(* PLC project Adressering.ecp, WAGO e!COCKPIT e!COCKPIT *)
(* stored: creationDateTime 2021-01-18T14:20:23.2110188, modificationDateTime 2021-01-18T11:51:27.6823754 *)

TYPE dtRomtype_11111111111111 : STRUCT
  RB601_V : BOOL;  (* Bevegelse *)
  RB601_HVAC : BOOL;  (* HVAC signal *)
  RT601_CT : REAL;  (* Rom temperatur *)
  RT601_SP_D : REAL;  (* Temperatur SP *)
  RT601_SP_S : REAL;  (* Temperatur SP standby *)
  RT601_SP_N : REAL;  (* Temperatur SP nattsenk *)
  RT601_SP_F : REAL;  (* Temperatur SP frostsikring *)
  RT601_CS : REAL;  (* Aktivt temperatur SP *)
  OPM : INT;  (* Rom modus *)
  OPM_CV : INT;  (* Rom modus verdi *)
  RY601_CV : REAL;  (* Co2 Nivaa *)
  RY601_SP : REAL;  (* Co2 SP *)
  RY601_OP : REAL;  (* Co2 paadrag *)
  LH601_OP : REAL;  (* Varmepaadrag *)
  LH601_MAN : BOOL;  (* Force LH *)
  LH601_CMD : BOOL;  (* LH601_CMD *)
  LC601_OP : REAL;  (* LC601_OP *)
  LC601_SP : REAL;  (* LC SP *)
  LC601_MAN : BOOL;  (* Force LC *)
  LC601_CMD : BOOL;  (* LC601_CMD *)
  RT601_SP : REAL;  (* Temperatur SP feedback *)
  RT601_SP_FB : REAL;  (* Temperatur SP *)
  RT601_SP_IN : REAL;  (* Temperatur SP lokalt panel *)
  LU601_V : BOOL;  (* Befukter status *)
  LU601_AL : BOOL;  (* Befukter alarm/feil *)
  LU601_CMD : BOOL;  (* Befukter tillat start *)
  OPM_001 : BYTE;  (* OPM output *)
END_STRUCT;
END_TYPE

TYPE dtRomtype_33333333333333 : STRUCT
  RB601_V : BOOL;  (* Bevegelse *)
  RB602_V : BOOL;  (* Bevegelse *)
  RB603_V : BOOL;  (* Bevegelse *)
  RB601_HVAC : BOOL;  (* HVAC signal *)
  RB602_HVAC : BOOL;  (* HVAC signal *)
  RB603_HVAC : BOOL;  (* HVAC signal *)
  RT601_CT : REAL;  (* Rom temperatur *)
  RT602_CT : REAL;  (* Rom temperatur *)
  RT602_SP : REAL;  (* Temperatur SP *)
  RT603_CT : REAL;  (* Rom temperatur *)
  RT603_SP : REAL;  (* Temperatur SP *)
  RT601_SP_D : REAL;  (* Temperatur SP *)
  RT601_SP_S : REAL;  (* Temperatur SP standby *)
  RT601_SP_N : REAL;  (* Temperatur SP nattsenk *)
  RT601_SP_F : REAL;  (* Temperatur SP frostsikring *)
  RT601_CS : REAL;  (* Aktivt temperatur SP *)
  OPM : INT;  (* Rom modus *)
  OPM_CV : INT;  (* Rom modus verdi *)
  RY601_CV : REAL;  (* Co2 Nivaa *)
  RY602_CV : REAL;  (* Co2 Nivaa *)
  RY603_CV : REAL;  (* Co2 Nivaa *)
  RY601_SP : REAL;  (* Co2 SP *)
  RY601_OP : REAL;  (* Co2 paadrag *)
  LH601_OP : REAL;  (* Varmepaadrag *)
  LH602_OP : REAL;  (* Varmepaadrag *)
  LH603_OP : REAL;  (* Varmepaadrag *)
  LH601_MAN : BOOL;  (* Force LH *)
  LH601_CMD : BOOL;  (* LH601_CMD *)
  LH602_CMD : BOOL;  (* LH602_CMD *)
  LH603_CMD : BOOL;  (* LH603_CMD *)
  LC601_OP : REAL;  (* LC601_OP *)
  LC602_OP : REAL;  (* LC602_OP *)
  LC603_OP : REAL;  (* LC603_OP *)
  LC601_SP : REAL;  (* LC SP *)
  LC601_MAN : BOOL;  (* Force LC *)
  LC601_CMD : BOOL;  (* LC601_CMD *)
  LC602_CMD : BOOL;  (* LC602_CMD *)
  LC603_CMD : BOOL;  (* LC603_CMD *)
  RT601_SP : REAL;  (* Temperatur SP feedback *)
  RT601_SP_FB : REAL;  (* Temperatur SP *)
  RT601_SP_IN : REAL;  (* Temperatur SP lokalt panel *)
  RT602_SP_FB : REAL;  (* Temperatur SP *)
  RT602_SP_IN : REAL;  (* Temperatur SP lokalt panel *)
  RT603_SP_FB : REAL;  (* Temperatur SP *)
  RT603_SP_IN : REAL;  (* Temperatur SP lokalt panel *)
  LU601_V : BOOL;  (* Befukter status *)
  LU602_V : BOOL;  (* Befukter status *)
  LU603_V : BOOL;  (* Befukter status *)
  LU601_AL : BOOL;  (* Befukter alarm/feil *)
  LU602_AL : BOOL;  (* Befukter alarm/feil *)
  LU603_AL : BOOL;  (* Befukter alarm/feil *)
  LU601_CMD : BOOL;  (* Befukter tillat start *)
  LU602_CMD : BOOL;  (* Befukter tillat start *)
  LU603_CMD : BOOL;  (* Befukter tillat start *)
  OPM_001 : BYTE;  (* OPM output *)
  OPM_002 : BYTE;  (* OPM output *)
  OPM_003 : BYTE;  (* OPM output *)
END_STRUCT;
END_TYPE

TYPE dtRomtype_99999999999999 : STRUCT
  RB601_V : BOOL;  (* Bevegelse *)
  RB602_V : BOOL;  (* Bevegelse *)
  RB603_V : BOOL;  (* Bevegelse *)
  RB604_V : BOOL;  (* Bevegelse *)
  RB605_V : BOOL;  (* Bevegelse *)
  RB606_V : BOOL;  (* Bevegelse *)
  RB607_V : BOOL;  (* Bevegelse *)
  RB608_V : BOOL;  (* Bevegelse *)
  RB609_V : BOOL;  (* Bevegelse *)
  RB601_HVAC : BOOL;  (* HVAC signal *)
  RB602_HVAC : BOOL;  (* HVAC signal *)
  RB603_HVAC : BOOL;  (* HVAC signal *)
  RB604_HVAC : BOOL;  (* HVAC signal *)
  RB605_HVAC : BOOL;  (* HVAC signal *)
  RB606_HVAC : BOOL;  (* HVAC signal *)
  RB607_HVAC : BOOL;  (* HVAC signal *)
  RB608_HVAC : BOOL;  (* HVAC signal *)
  RB609_HVAC : BOOL;  (* HVAC signal *)
  RT601_CT : REAL;  (* Rom temperatur *)
  RT602_CT : REAL;  (* Rom temperatur *)
  RT602_SP : REAL;  (* Temperatur SP *)
  RT603_CT : REAL;  (* Rom temperatur *)
  RT603_SP : REAL;  (* Temperatur SP *)
  RT604_CT : REAL;  (* Rom temperatur *)
  RT604_SP : REAL;  (* Temperatur SP *)
  RT605_CT : REAL;  (* Rom temperatur *)
  RT605_SP : REAL;  (* Temperatur SP *)
  RT606_CT : REAL;  (* Rom temperatur *)
  RT606_SP : REAL;  (* Temperatur SP *)
  RT607_CT : REAL;  (* Rom temperatur *)
  RT607_SP : REAL;  (* Temperatur SP *)
  RT608_CT : REAL;  (* Rom temperatur *)
  RT608_SP : REAL;  (* Temperatur SP *)
  RT609_CT : REAL;  (* Rom temperatur *)
  RT609_SP : REAL;  (* Temperatur SP *)
  RT601_SP_D : REAL;  (* Temperatur SP *)
  RT601_SP_S : REAL;  (* Temperatur SP standby *)
  RT601_SP_N : REAL;  (* Temperatur SP nattsenk *)
  RT601_SP_F : REAL;  (* Temperatur SP frostsikring *)
  RT601_CS : REAL;  (* Aktivt temperatur SP *)
  OPM : INT;  (* Rom modus *)
  OPM_CV : INT;  (* Rom modus verdi *)
  RY601_CV : REAL;  (* Co2 Nivaa *)
  RY602_CV : REAL;  (* Co2 Nivaa *)
  RY603_CV : REAL;  (* Co2 Nivaa *)
  RY604_CV : REAL;  (* Co2 Nivaa *)
  RY605_CV : REAL;  (* Co2 Nivaa *)
  RY606_CV : REAL;  (* Co2 Nivaa *)
  RY607_CV : REAL;  (* Co2 Nivaa *)
  RY608_CV : REAL;  (* Co2 Nivaa *)
  RY609_CV : REAL;  (* Co2 Nivaa *)
  RY601_SP : REAL;  (* Co2 SP *)
  RY601_OP : REAL;  (* Co2 paadrag *)
  LH601_OP : REAL;  (* Varmepaadrag *)
  LH602_OP : REAL;  (* Varmepaadrag *)
  LH603_OP : REAL;  (* Varmepaadrag *)
  LH604_OP : REAL;  (* Varmepaadrag *)
  LH605_OP : REAL;  (* Varmepaadrag *)
  LH606_OP : REAL;  (* Varmepaadrag *)
  LH607_OP : REAL;  (* Varmepaadrag *)
  LH608_OP : REAL;  (* Varmepaadrag *)
  LH609_OP : REAL;  (* Varmepaadrag *)
  LH601_MAN : BOOL;  (* Force LH *)
  LH601_CMD : BOOL;  (* LH601_CMD *)
  LH602_CMD : BOOL;  (* LH602_CMD *)
  LH603_CMD : BOOL;  (* LH603_CMD *)
  LH604_CMD : BOOL;  (* LH604_CMD *)
  LH605_CMD : BOOL;  (* LH605_CMD *)
  LH606_CMD : BOOL;  (* LH606_CMD *)
  LH607_CMD : BOOL;  (* LH607_CMD *)
  LH608_CMD : BOOL;  (* LH608_CMD *)
  LH609_CMD : BOOL;  (* LH609_CMD *)
  LC601_OP : REAL;  (* LC601_OP *)
  LC602_OP : REAL;  (* LC602_OP *)
  LC603_OP : REAL;  (* LC603_OP *)
  LC604_OP : REAL;  (* LC604_OP *)
  LC605_OP : REAL;  (* LC605_OP *)
  LC606_OP : REAL;  (* LC606_OP *)
  LC607_OP : REAL;  (* LC607_OP *)
  LC608_OP : REAL;  (* LC608_OP *)
  LC609_OP : REAL;  (* LC609_OP *)
  LC601_SP : REAL;  (* LC SP *)
  LC601_MAN : BOOL;  (* Force LC *)
  LC601_CMD : BOOL;  (* LC601_CMD *)
  LC602_CMD : BOOL;  (* LC602_CMD *)
  LC603_CMD : BOOL;  (* LC603_CMD *)
  LC604_CMD : BOOL;  (* LC604_CMD *)
  LC605_CMD : BOOL;  (* LC605_CMD *)
  LC606_CMD : BOOL;  (* LC606_CMD *)
  LC607_CMD : BOOL;  (* LC607_CMD *)
  LC608_CMD : BOOL;  (* LC608_CMD *)
  LC609_CMD : BOOL;  (* LC609_CMD *)
  RT601_SP : REAL;  (* Temperatur SP feedback *)
  RT601_SP_FB : REAL;  (* Temperatur SP *)
  RT601_SP_IN : REAL;  (* Temperatur SP lokalt panel *)
  RT602_SP_FB : REAL;  (* Temperatur SP *)
  RT602_SP_IN : REAL;  (* Temperatur SP lokalt panel *)
  RT603_SP_FB : REAL;  (* Temperatur SP *)
  RT603_SP_IN : REAL;  (* Temperatur SP lokalt panel *)
  RT604_SP_FB : REAL;  (* Temperatur SP *)
  RT604_SP_IN : REAL;  (* Temperatur SP lokalt panel *)
  RT605_SP_FB : REAL;  (* Temperatur SP *)
  RT605_SP_IN : REAL;  (* Temperatur SP lokalt panel *)
  RT606_SP_FB : REAL;  (* Temperatur SP *)
  RT606_SP_IN : REAL;  (* Temperatur SP lokalt panel *)
  RT607_SP_FB : REAL;  (* Temperatur SP *)
  RT607_SP_IN : REAL;  (* Temperatur SP lokalt panel *)
  RT608_SP_FB : REAL;  (* Temperatur SP *)
  RT608_SP_IN : REAL;  (* Temperatur SP lokalt panel *)
  RT609_SP_FB : REAL;  (* Temperatur SP *)
  RT609_SP_IN : REAL;  (* Temperatur SP lokalt panel *)
  LU601_V : BOOL;  (* Befukter status *)
  LU602_V : BOOL;  (* Befukter status *)
  LU603_V : BOOL;  (* Befukter status *)
  LU604_V : BOOL;  (* Befukter status *)
  LU605_V : BOOL;  (* Befukter status *)
  LU606_V : BOOL;  (* Befukter status *)
  LU607_V : BOOL;  (* Befukter status *)
  LU608_V : BOOL;  (* Befukter status *)
  LU609_V : BOOL;  (* Befukter status *)
  LU601_AL : BOOL;  (* Befukter alarm/feil *)
  LU602_AL : BOOL;  (* Befukter alarm/feil *)
  LU603_AL : BOOL;  (* Befukter alarm/feil *)
  LU604_AL : BOOL;  (* Befukter alarm/feil *)
  LU605_AL : BOOL;  (* Befukter alarm/feil *)
  LU606_AL : BOOL;  (* Befukter alarm/feil *)
  LU607_AL : BOOL;  (* Befukter alarm/feil *)
  LU608_AL : BOOL;  (* Befukter alarm/feil *)
  LU609_AL : BOOL;  (* Befukter alarm/feil *)
  LU601_CMD : BOOL;  (* Befukter tillat start *)
  LU602_CMD : BOOL;  (* Befukter tillat start *)
  LU603_CMD : BOOL;  (* Befukter tillat start *)
  LU604_CMD : BOOL;  (* Befukter tillat start *)
  LU605_CMD : BOOL;  (* Befukter tillat start *)
  LU606_CMD : BOOL;  (* Befukter tillat start *)
  LU607_CMD : BOOL;  (* Befukter tillat start *)
  LU608_CMD : BOOL;  (* Befukter tillat start *)
  LU609_CMD : BOOL;  (* Befukter tillat start *)
  OPM_001 : BYTE;  (* OPM output *)
  OPM_002 : BYTE;  (* OPM output *)
  OPM_003 : BYTE;  (* OPM output *)
  OPM_004 : BYTE;  (* OPM output *)
  OPM_005 : BYTE;  (* OPM output *)
  OPM_006 : BYTE;  (* OPM output *)
  OPM_007 : BYTE;  (* OPM output *)
  OPM_008 : BYTE;  (* OPM output *)
  OPM_009 : BYTE;  (* OPM output *)
END_STRUCT;
END_TYPE

{attribute 'qualified_only'}
VAR_GLOBAL  (* STLV59_563 *)
  STLV59_A_563_RB001_HVAC : BOOL;  (* HVAC signal for PLS *)
  STLV59_A_563_KNX_Card_1_Status : BOOL;  (* KNX kort 1 status *)
  STLV59_A_563_001 : dtRomtype_11111111111111;  (* Placeholder_1 *)
  STLV59_A_563_002 : dtRomtype_33333333333333;  (* Placeholder_2 *)
  STLV59_A_563_003 : dtRomtype_99999999999999;  (* Placeholder_3 *)
END_VAR

FUNCTION_BLOCK fbRomtype_11111111111111
  VAR_INPUT
    RB601_HVAC : BOOL;
    RT601_CT : REAL;
    RT601_SP_D : REAL;
    RT601_SP_S : REAL;
    RT601_SP_N : REAL;
    RT601_SP_F : REAL;
    OPM : INT;
    RY601_CV : REAL;
    RY601_SP : REAL;
    LH601_MAN : BOOL;
    LC601_SP : REAL;
    LC601_MAN : BOOL;
    RT601_SP_IN : REAL;
    LU601_V : BOOL;
  END_VAR
  VAR_OUTPUT
    OPM_CV : INT;
    RT601_CS : REAL;
    RY601_OP : REAL;
    LH601_OP : REAL;
    LH601_CMD : BOOL;
    LC601_OP : REAL;
    LC601_CMD : BOOL;
    LU601_CMD : BOOL;
    OPM_001 : BYTE;
  END_VAR

(* CFC diagram, written out as Structured Text *)
END_FUNCTION_BLOCK

FUNCTION_BLOCK fbRomtype_33333333333333
  VAR_INPUT
    RB601_HVAC : BOOL;
    RB602_HVAC : BOOL;
    RB603_HVAC : BOOL;
    RT601_CT : REAL;
    RT602_CT : REAL;
    RT602_SP : REAL;
    RT603_CT : REAL;
    RT603_SP : REAL;
    RT601_SP_D : REAL;
    RT601_SP_S : REAL;
    RT601_SP_N : REAL;
    RT601_SP_F : REAL;
    OPM : INT;
    RY601_CV : REAL;
    RY602_CV : REAL;
    RY603_CV : REAL;
    RY601_SP : REAL;
    LH601_MAN : BOOL;
    LC601_SP : REAL;
    LC601_MAN : BOOL;
    RT601_SP_IN : REAL;
    RT602_SP_IN : REAL;
    RT603_SP_IN : REAL;
    LU601_V : BOOL;
    LU602_V : BOOL;
    LU603_V : BOOL;
  END_VAR
  VAR_OUTPUT
    OPM_CV : INT;
    RT601_CS : REAL;
    RT602_CS : REAL;
    RT603_CS : REAL;
    RY601_OP : REAL;
    LH601_OP : REAL;
    LH602_OP : REAL;
    LH603_OP : REAL;
    LH601_CMD : BOOL;
    LH602_CMD : BOOL;
    LH603_CMD : BOOL;
    LC601_OP : REAL;
    LC602_OP : REAL;
    LC603_OP : REAL;
    LC601_CMD : BOOL;
    LC602_CMD : BOOL;
    LC603_CMD : BOOL;
    LU601_CMD : BOOL;
    LU602_CMD : BOOL;
    LU603_CMD : BOOL;
    OPM_001 : BYTE;
    OPM_002 : BYTE;
    OPM_003 : BYTE;
  END_VAR

(* CFC diagram, written out as Structured Text *)
END_FUNCTION_BLOCK

FUNCTION_BLOCK fbRomtype_99999999999999
  VAR_INPUT
    RB601_HVAC : BOOL;
    RB602_HVAC : BOOL;
    RB603_HVAC : BOOL;
    RB604_HVAC : BOOL;
    RB605_HVAC : BOOL;
    RB606_HVAC : BOOL;
    RB607_HVAC : BOOL;
    RB608_HVAC : BOOL;
    RB609_HVAC : BOOL;
    RT601_CT : REAL;
    RT602_CT : REAL;
    RT602_SP : REAL;
    RT603_CT : REAL;
    RT603_SP : REAL;
    RT604_CT : REAL;
    RT604_SP : REAL;
    RT605_CT : REAL;
    RT605_SP : REAL;
    RT606_CT : REAL;
    RT606_SP : REAL;
    RT607_CT : REAL;
    RT607_SP : REAL;
    RT608_CT : REAL;
    RT608_SP : REAL;
    RT609_CT : REAL;
    RT609_SP : REAL;
    RT601_SP_D : REAL;
    RT601_SP_S : REAL;
    RT601_SP_N : REAL;
    RT601_SP_F : REAL;
    OPM : INT;
    RY601_CV : REAL;
    RY602_CV : REAL;
    RY603_CV : REAL;
    RY604_CV : REAL;
    RY605_CV : REAL;
    RY606_CV : REAL;
    RY607_CV : REAL;
    RY608_CV : REAL;
    RY609_CV : REAL;
    RY601_SP : REAL;
    LH601_MAN : BOOL;
    LC601_SP : REAL;
    LC601_MAN : BOOL;
    RT601_SP_IN : REAL;
    RT602_SP_IN : REAL;
    RT603_SP_IN : REAL;
    RT604_SP_IN : REAL;
    RT605_SP_IN : REAL;
    RT606_SP_IN : REAL;
    RT607_SP_IN : REAL;
    RT608_SP_IN : REAL;
    RT609_SP_IN : REAL;
    LU601_V : BOOL;
    LU602_V : BOOL;
    LU603_V : BOOL;
    LU604_V : BOOL;
    LU605_V : BOOL;
    LU606_V : BOOL;
    LU607_V : BOOL;
    LU608_V : BOOL;
    LU609_V : BOOL;
  END_VAR
  VAR_OUTPUT
    OPM_CV : INT;
    RT601_CS : REAL;
    RT602_CS : REAL;
    RT603_CS : REAL;
    RT604_CS : REAL;
    RT605_CS : REAL;
    RT606_CS : REAL;
    RT607_CS : REAL;
    RT608_CS : REAL;
    RT609_CS : REAL;
    RY601_OP : REAL;
    LH601_OP : REAL;
    LH602_OP : REAL;
    LH603_OP : REAL;
    LH604_OP : REAL;
    LH605_OP : REAL;
    LH606_OP : REAL;
    LH607_OP : REAL;
    LH608_OP : REAL;
    LH609_OP : REAL;
    LH601_CMD : BOOL;
    LH602_CMD : BOOL;
    LH603_CMD : BOOL;
    LH604_CMD : BOOL;
    LH605_CMD : BOOL;
    LH606_CMD : BOOL;
    LH607_CMD : BOOL;
    LH608_CMD : BOOL;
    LH609_CMD : BOOL;
    LC601_OP : REAL;
    LC602_OP : REAL;
    LC603_OP : REAL;
    LC604_OP : REAL;
    LC605_OP : REAL;
    LC606_OP : REAL;
    LC607_OP : REAL;
    LC608_OP : REAL;
    LC609_OP : REAL;
    LC601_CMD : BOOL;
    LC602_CMD : BOOL;
    LC603_CMD : BOOL;
    LC604_CMD : BOOL;
    LC605_CMD : BOOL;
    LC606_CMD : BOOL;
    LC607_CMD : BOOL;
    LC608_CMD : BOOL;
    LC609_CMD : BOOL;
    LU601_CMD : BOOL;
    LU602_CMD : BOOL;
    LU603_CMD : BOOL;
    LU604_CMD : BOOL;
    LU605_CMD : BOOL;
    LU606_CMD : BOOL;
    LU607_CMD : BOOL;
    LU608_CMD : BOOL;
    LU609_CMD : BOOL;
    OPM_001 : BYTE;
    OPM_002 : BYTE;
    OPM_003 : BYTE;
    OPM_004 : BYTE;
    OPM_005 : BYTE;
    OPM_006 : BYTE;
    OPM_007 : BYTE;
    OPM_008 : BYTE;
    OPM_009 : BYTE;
  END_VAR

(* CFC diagram, written out as Structured Text *)
END_FUNCTION_BLOCK

PROGRAM PRG_KNX_563_1
  VAR
    i : INT := 0;  (* Felles *)
    Interval : TON := (PT := TIME#2m0s0ms);
    typDPT : typDPT;
    KNX_master_1 : WagoAppKNX.FbKNX_Master;  (* Master *)
    M1_001_001_RB601_V : fbDPT_Switch_pro;  (* 001 *)
    M1_002_001_RB601_HVAC : fbDPT_Switch_pro;
    M1_003_001_RT601_CT : fbDPT_Value_Temp_pro;
    M1_004_001_RY601_CV : fbDPT_Value_AirQuality_pro;
    M1_005_001_LH601_OP : fbDPT_Scaling_pro;
    M1_006_001_LH601_CMD : fbDPT_Switch_pro;
    M1_007_001_LC601_OP : fbDPT_Scaling_pro;
    M1_008_001_LC601_CMD : fbDPT_Switch_pro;
    M1_009_001_RT601_SP : fbDPT_Value_Temp_pro;
    M1_010_001_RT601_SP_FB : fbDPT_Value_Temp_pro;
    M1_011_001_LU601_V : fbDPT_Switch_pro;
    M1_012_001_LU601_AL : fbDPT_Switch_pro;
    M1_013_001_LU601_CMD : fbDPT_Switch_pro;
    M1_014_001_OPM_001 : fbDPT_1_BYTE;
    M1_015_002_RB601_V : fbDPT_Switch_pro;  (* 002 *)
    M1_016_002_RB602_V : fbDPT_Switch_pro;
    M1_017_002_RB603_V : fbDPT_Switch_pro;
    M1_018_002_RB601_HVAC : fbDPT_Switch_pro;
    M1_019_002_RB602_HVAC : fbDPT_Switch_pro;
    M1_020_002_RB603_HVAC : fbDPT_Switch_pro;
    M1_021_002_RT601_CT : fbDPT_Value_Temp_pro;
    M1_022_002_RT602_CT : fbDPT_Value_Temp_pro;
    M1_023_002_RT603_CT : fbDPT_Value_Temp_pro;
    M1_024_002_RY601_CV : fbDPT_Value_AirQuality_pro;
    M1_025_002_RY602_CV : fbDPT_Value_AirQuality_pro;
    M1_026_002_RY603_CV : fbDPT_Value_AirQuality_pro;
    M1_027_002_LH601_OP : fbDPT_Scaling_pro;
    M1_028_002_LH602_OP : fbDPT_Scaling_pro;
    M1_029_002_LH603_OP : fbDPT_Scaling_pro;
    M1_030_002_LH601_CMD : fbDPT_Switch_pro;
    M1_031_002_LH602_CMD : fbDPT_Switch_pro;
    M1_032_002_LH603_CMD : fbDPT_Switch_pro;
    M1_033_002_LC601_OP : fbDPT_Scaling_pro;
    M1_034_002_LC602_OP : fbDPT_Scaling_pro;
    M1_035_002_LC603_OP : fbDPT_Scaling_pro;
    M1_036_002_LC601_CMD : fbDPT_Switch_pro;
    M1_037_002_LC602_CMD : fbDPT_Switch_pro;
    M1_038_002_LC603_CMD : fbDPT_Switch_pro;
    M1_039_002_RT601_SP : fbDPT_Value_Temp_pro;
    M1_040_002_RT602_SP : fbDPT_Value_Temp_pro;
    M1_041_002_RT603_SP : fbDPT_Value_Temp_pro;
    M1_042_002_RT601_SP_FB : fbDPT_Value_Temp_pro;
    M1_043_002_RT602_SP_FB : fbDPT_Value_Temp_pro;
    M1_044_002_RT603_SP_FB : fbDPT_Value_Temp_pro;
    M1_045_002_LU601_V : fbDPT_Switch_pro;
    M1_046_002_LU602_V : fbDPT_Switch_pro;
    M1_047_002_LU603_V : fbDPT_Switch_pro;
    M1_048_002_LU601_AL : fbDPT_Switch_pro;
    M1_049_002_LU602_AL : fbDPT_Switch_pro;
    M1_050_002_LU603_AL : fbDPT_Switch_pro;
    M1_051_002_LU601_CMD : fbDPT_Switch_pro;
    M1_052_002_LU602_CMD : fbDPT_Switch_pro;
    M1_053_002_LU603_CMD : fbDPT_Switch_pro;
    M1_054_002_OPM_001 : fbDPT_1_BYTE;
    M1_055_002_OPM_002 : fbDPT_1_BYTE;
    M1_056_002_OPM_003 : fbDPT_1_BYTE;
    M1_057_003_RB601_V : fbDPT_Switch_pro;  (* 003 *)
    M1_058_003_RB602_V : fbDPT_Switch_pro;
    M1_059_003_RB603_V : fbDPT_Switch_pro;
    M1_060_003_RB604_V : fbDPT_Switch_pro;
    M1_061_003_RB605_V : fbDPT_Switch_pro;
    M1_062_003_RB606_V : fbDPT_Switch_pro;
    M1_063_003_RB607_V : fbDPT_Switch_pro;
    M1_064_003_RB608_V : fbDPT_Switch_pro;
    M1_065_003_RB609_V : fbDPT_Switch_pro;
    M1_066_003_RB601_HVAC : fbDPT_Switch_pro;
    M1_067_003_RB602_HVAC : fbDPT_Switch_pro;
    M1_068_003_RB603_HVAC : fbDPT_Switch_pro;
    M1_069_003_RB604_HVAC : fbDPT_Switch_pro;
    M1_070_003_RB605_HVAC : fbDPT_Switch_pro;
    M1_071_003_RB606_HVAC : fbDPT_Switch_pro;
    M1_072_003_RB607_HVAC : fbDPT_Switch_pro;
    M1_073_003_RB608_HVAC : fbDPT_Switch_pro;
    M1_074_003_RB609_HVAC : fbDPT_Switch_pro;
    M1_075_003_RT601_CT : fbDPT_Value_Temp_pro;
    M1_076_003_RT602_CT : fbDPT_Value_Temp_pro;
    M1_077_003_RT603_CT : fbDPT_Value_Temp_pro;
    M1_078_003_RT604_CT : fbDPT_Value_Temp_pro;
    M1_079_003_RT605_CT : fbDPT_Value_Temp_pro;
    M1_080_003_RT606_CT : fbDPT_Value_Temp_pro;
    M1_081_003_RT607_CT : fbDPT_Value_Temp_pro;
    M1_082_003_RT608_CT : fbDPT_Value_Temp_pro;
    M1_083_003_RT609_CT : fbDPT_Value_Temp_pro;
    M1_084_003_RY601_CV : fbDPT_Value_AirQuality_pro;
    M1_085_003_RY602_CV : fbDPT_Value_AirQuality_pro;
    M1_086_003_RY603_CV : fbDPT_Value_AirQuality_pro;
    M1_087_003_RY604_CV : fbDPT_Value_AirQuality_pro;
    M1_088_003_RY605_CV : fbDPT_Value_AirQuality_pro;
    M1_089_003_RY606_CV : fbDPT_Value_AirQuality_pro;
    M1_090_003_RY607_CV : fbDPT_Value_AirQuality_pro;
    M1_091_003_RY608_CV : fbDPT_Value_AirQuality_pro;
    M1_092_003_RY609_CV : fbDPT_Value_AirQuality_pro;
    M1_093_003_LH601_OP : fbDPT_Scaling_pro;
    M1_094_003_LH602_OP : fbDPT_Scaling_pro;
    M1_095_003_LH603_OP : fbDPT_Scaling_pro;
    M1_096_003_LH604_OP : fbDPT_Scaling_pro;
    M1_097_003_LH605_OP : fbDPT_Scaling_pro;
    M1_098_003_LH606_OP : fbDPT_Scaling_pro;
    M1_099_003_LH607_OP : fbDPT_Scaling_pro;
    M1_0100_003_LH608_OP : fbDPT_Scaling_pro;
    M1_0101_003_LH609_OP : fbDPT_Scaling_pro;
    M1_102_003_LH601_CMD : fbDPT_Switch_pro;
    M1_103_003_LH602_CMD : fbDPT_Switch_pro;
    M1_104_003_LH603_CMD : fbDPT_Switch_pro;
    M1_105_003_LH604_CMD : fbDPT_Switch_pro;
    M1_106_003_LH605_CMD : fbDPT_Switch_pro;
    M1_107_003_LH606_CMD : fbDPT_Switch_pro;
    M1_108_003_LH607_CMD : fbDPT_Switch_pro;
    M1_109_003_LH608_CMD : fbDPT_Switch_pro;
    M1_110_003_LH609_CMD : fbDPT_Switch_pro;
    M1_111_003_LC601_OP : fbDPT_Scaling_pro;
    M1_112_003_LC602_OP : fbDPT_Scaling_pro;
    M1_113_003_LC603_OP : fbDPT_Scaling_pro;
    M1_114_003_LC604_OP : fbDPT_Scaling_pro;
    M1_115_003_LC605_OP : fbDPT_Scaling_pro;
    M1_116_003_LC606_OP : fbDPT_Scaling_pro;
    M1_117_003_LC607_OP : fbDPT_Scaling_pro;
    M1_118_003_LC608_OP : fbDPT_Scaling_pro;
    M1_119_003_LC609_OP : fbDPT_Scaling_pro;
    M1_120_003_LC601_CMD : fbDPT_Switch_pro;
    M1_121_003_LC602_CMD : fbDPT_Switch_pro;
    M1_122_003_LC603_CMD : fbDPT_Switch_pro;
    M1_123_003_LC604_CMD : fbDPT_Switch_pro;
    M1_124_003_LC605_CMD : fbDPT_Switch_pro;
    M1_125_003_LC606_CMD : fbDPT_Switch_pro;
    M1_126_003_LC607_CMD : fbDPT_Switch_pro;
    M1_127_003_LC608_CMD : fbDPT_Switch_pro;
    M1_128_003_LC609_CMD : fbDPT_Switch_pro;
    M1_129_003_RT601_SP : fbDPT_Value_Temp_pro;
    M1_130_003_RT602_SP : fbDPT_Value_Temp_pro;
    M1_131_003_RT603_SP : fbDPT_Value_Temp_pro;
    M1_132_003_RT604_SP : fbDPT_Value_Temp_pro;
    M1_133_003_RT605_SP : fbDPT_Value_Temp_pro;
    M1_134_003_RT606_SP : fbDPT_Value_Temp_pro;
    M1_135_003_RT607_SP : fbDPT_Value_Temp_pro;
    M1_136_003_RT608_SP : fbDPT_Value_Temp_pro;
    M1_137_003_RT609_SP : fbDPT_Value_Temp_pro;
    M1_138_003_RT601_SP_FB : fbDPT_Value_Temp_pro;
    M1_139_003_RT602_SP_FB : fbDPT_Value_Temp_pro;
    M1_140_003_RT603_SP_FB : fbDPT_Value_Temp_pro;
    M1_141_003_RT604_SP_FB : fbDPT_Value_Temp_pro;
    M1_142_003_RT605_SP_FB : fbDPT_Value_Temp_pro;
    M1_143_003_RT606_SP_FB : fbDPT_Value_Temp_pro;
    M1_144_003_RT607_SP_FB : fbDPT_Value_Temp_pro;
    M1_145_003_RT608_SP_FB : fbDPT_Value_Temp_pro;
    M1_146_003_RT609_SP_FB : fbDPT_Value_Temp_pro;
    M1_147_003_LU601_V : fbDPT_Switch_pro;
    M1_148_003_LU602_V : fbDPT_Switch_pro;
    M1_149_003_LU603_V : fbDPT_Switch_pro;
    M1_150_003_LU604_V : fbDPT_Switch_pro;
    M1_151_003_LU605_V : fbDPT_Switch_pro;
    M1_152_003_LU606_V : fbDPT_Switch_pro;
    M1_153_003_LU607_V : fbDPT_Switch_pro;
    M1_154_003_LU608_V : fbDPT_Switch_pro;
    M1_155_003_LU609_V : fbDPT_Switch_pro;
    M1_156_003_LU601_AL : fbDPT_Switch_pro;
    M1_157_003_LU602_AL : fbDPT_Switch_pro;
    M1_158_003_LU603_AL : fbDPT_Switch_pro;
    M1_159_003_LU604_AL : fbDPT_Switch_pro;
    M1_160_003_LU605_AL : fbDPT_Switch_pro;
    M1_161_003_LU606_AL : fbDPT_Switch_pro;
    M1_162_003_LU607_AL : fbDPT_Switch_pro;
    M1_163_003_LU608_AL : fbDPT_Switch_pro;
    M1_164_003_LU609_AL : fbDPT_Switch_pro;
    M1_165_003_LU601_CMD : fbDPT_Switch_pro;
    M1_166_003_LU602_CMD : fbDPT_Switch_pro;
    M1_167_003_LU603_CMD : fbDPT_Switch_pro;
    M1_168_003_LU604_CMD : fbDPT_Switch_pro;
    M1_169_003_LU605_CMD : fbDPT_Switch_pro;
    M1_170_003_LU606_CMD : fbDPT_Switch_pro;
    M1_171_003_LU607_CMD : fbDPT_Switch_pro;
    M1_172_003_LU608_CMD : fbDPT_Switch_pro;
    M1_173_003_LU609_CMD : fbDPT_Switch_pro;
    M1_174_003_OPM_001 : fbDPT_1_BYTE;
    M1_175_003_OPM_002 : fbDPT_1_BYTE;
    M1_176_003_OPM_003 : fbDPT_1_BYTE;
    M1_177_003_OPM_004 : fbDPT_1_BYTE;
    M1_178_003_OPM_005 : fbDPT_1_BYTE;
    M1_179_003_OPM_006 : fbDPT_1_BYTE;
    M1_180_003_OPM_007 : fbDPT_1_BYTE;
    M1_181_003_OPM_008 : fbDPT_1_BYTE;
    M1_182_003_OPM_009 : fbDPT_1_BYTE;
  END_VAR
  VAR  (* added by the conversion: wires and edge detectors of the diagram *)
    _ADD9_OUT : INT;
    _GT15_OUT : BOOL;
    _MOVE19_ENO : BOOL;
    _MOVE19_OUT : INT;
    _MOVE46_ENO : BOOL;
    _MOVE46_OUT : ANY;
    _MOVE59_ENO : BOOL;
    _MOVE59_OUT : ANY;
    _MOVE72_ENO : BOOL;
    _MOVE72_OUT : ANY;
    _MOVE85_ENO : BOOL;
    _MOVE85_OUT : ANY;
    _MOVE174_ENO : BOOL;
    _MOVE174_OUT : ANY;
    _MOVE187_ENO : BOOL;
    _MOVE187_OUT : ANY;
    _MOVE200_ENO : BOOL;
    _MOVE200_OUT : ANY;
    _MOVE246_ENO : BOOL;
    _MOVE246_OUT : ANY;
    _MOVE259_ENO : BOOL;
    _MOVE259_OUT : ANY;
    _MOVE272_ENO : BOOL;
    _MOVE272_OUT : ANY;
    _MOVE285_ENO : BOOL;
    _MOVE285_OUT : ANY;
    _MOVE298_ENO : BOOL;
    _MOVE298_OUT : ANY;
    _MOVE311_ENO : BOOL;
    _MOVE311_OUT : ANY;
    _MOVE324_ENO : BOOL;
    _MOVE324_OUT : ANY;
    _MOVE337_ENO : BOOL;
    _MOVE337_OUT : ANY;
    _MOVE350_ENO : BOOL;
    _MOVE350_OUT : ANY;
    _MOVE363_ENO : BOOL;
    _MOVE363_OUT : ANY;
    _MOVE376_ENO : BOOL;
    _MOVE376_OUT : ANY;
    _MOVE389_ENO : BOOL;
    _MOVE389_OUT : ANY;
    _MOVE630_ENO : BOOL;
    _MOVE630_OUT : ANY;
    _MOVE643_ENO : BOOL;
    _MOVE643_OUT : ANY;
    _MOVE656_ENO : BOOL;
    _MOVE656_OUT : ANY;
    _MOVE669_ENO : BOOL;
    _MOVE669_OUT : ANY;
    _MOVE682_ENO : BOOL;
    _MOVE682_OUT : ANY;
    _MOVE695_ENO : BOOL;
    _MOVE695_OUT : ANY;
    _MOVE708_ENO : BOOL;
    _MOVE708_OUT : ANY;
    _MOVE721_ENO : BOOL;
    _MOVE721_OUT : ANY;
    _MOVE734_ENO : BOOL;
    _MOVE734_OUT : ANY;
    _MOVE844_ENO : BOOL;
    _MOVE844_OUT : ANY;
    _MOVE857_ENO : BOOL;
    _MOVE857_OUT : ANY;
    _MOVE870_ENO : BOOL;
    _MOVE870_OUT : ANY;
    _MOVE883_ENO : BOOL;
    _MOVE883_OUT : ANY;
    _MOVE896_ENO : BOOL;
    _MOVE896_OUT : ANY;
    _MOVE909_ENO : BOOL;
    _MOVE909_OUT : ANY;
    _MOVE922_ENO : BOOL;
    _MOVE922_OUT : ANY;
    _MOVE935_ENO : BOOL;
    _MOVE935_OUT : ANY;
    _MOVE948_ENO : BOOL;
    _MOVE948_OUT : ANY;
    _MOVE961_ENO : BOOL;
    _MOVE961_OUT : ANY;
    _MOVE974_ENO : BOOL;
    _MOVE974_OUT : ANY;
    _MOVE987_ENO : BOOL;
    _MOVE987_OUT : ANY;
    _MOVE1000_ENO : BOOL;
    _MOVE1000_OUT : ANY;
    _MOVE1013_ENO : BOOL;
    _MOVE1013_OUT : ANY;
    _MOVE1026_ENO : BOOL;
    _MOVE1026_OUT : ANY;
    _MOVE1039_ENO : BOOL;
    _MOVE1039_OUT : ANY;
    _MOVE1052_ENO : BOOL;
    _MOVE1052_OUT : ANY;
    _MOVE1065_ENO : BOOL;
    _MOVE1065_OUT : ANY;
    _MOVE1078_ENO : BOOL;
    _MOVE1078_OUT : ANY;
    _MOVE1091_ENO : BOOL;
    _MOVE1091_OUT : ANY;
    _MOVE1104_ENO : BOOL;
    _MOVE1104_OUT : ANY;
    _MOVE1117_ENO : BOOL;
    _MOVE1117_OUT : ANY;
    _MOVE1130_ENO : BOOL;
    _MOVE1130_OUT : ANY;
    _MOVE1143_ENO : BOOL;
    _MOVE1143_OUT : ANY;
    _MOVE1156_ENO : BOOL;
    _MOVE1156_OUT : ANY;
    _MOVE1169_ENO : BOOL;
    _MOVE1169_OUT : ANY;
    _MOVE1182_ENO : BOOL;
    _MOVE1182_OUT : ANY;
    _MOVE1195_ENO : BOOL;
    _MOVE1195_OUT : ANY;
    _MOVE1208_ENO : BOOL;
    _MOVE1208_OUT : ANY;
    _MOVE1221_ENO : BOOL;
    _MOVE1221_OUT : ANY;
    _MOVE1234_ENO : BOOL;
    _MOVE1234_OUT : ANY;
    _MOVE1247_ENO : BOOL;
    _MOVE1247_OUT : ANY;
    _MOVE1260_ENO : BOOL;
    _MOVE1260_OUT : ANY;
    _MOVE1273_ENO : BOOL;
    _MOVE1273_OUT : ANY;
    _MOVE1286_ENO : BOOL;
    _MOVE1286_OUT : ANY;
    _MOVE1299_ENO : BOOL;
    _MOVE1299_OUT : ANY;
    _MOVE1996_ENO : BOOL;
    _MOVE1996_OUT : ANY;
    _MOVE2009_ENO : BOOL;
    _MOVE2009_OUT : ANY;
    _MOVE2022_ENO : BOOL;
    _MOVE2022_OUT : ANY;
    _MOVE2035_ENO : BOOL;
    _MOVE2035_OUT : ANY;
    _MOVE2048_ENO : BOOL;
    _MOVE2048_OUT : ANY;
    _MOVE2061_ENO : BOOL;
    _MOVE2061_OUT : ANY;
    _MOVE2074_ENO : BOOL;
    _MOVE2074_OUT : ANY;
    _MOVE2087_ENO : BOOL;
    _MOVE2087_OUT : ANY;
    _MOVE2100_ENO : BOOL;
    _MOVE2100_OUT : ANY;
    _MOVE2113_ENO : BOOL;
    _MOVE2113_OUT : ANY;
    _MOVE2126_ENO : BOOL;
    _MOVE2126_OUT : ANY;
    _MOVE2139_ENO : BOOL;
    _MOVE2139_OUT : ANY;
    _MOVE2152_ENO : BOOL;
    _MOVE2152_OUT : ANY;
    _MOVE2165_ENO : BOOL;
    _MOVE2165_OUT : ANY;
    _MOVE2178_ENO : BOOL;
    _MOVE2178_OUT : ANY;
    _MOVE2191_ENO : BOOL;
    _MOVE2191_OUT : ANY;
    _MOVE2204_ENO : BOOL;
    _MOVE2204_OUT : ANY;
    _MOVE2217_ENO : BOOL;
    _MOVE2217_OUT : ANY;
    _MOVE2230_ENO : BOOL;
    _MOVE2230_OUT : ANY;
    _MOVE2243_ENO : BOOL;
    _MOVE2243_OUT : ANY;
    _MOVE2256_ENO : BOOL;
    _MOVE2256_OUT : ANY;
    _MOVE2269_ENO : BOOL;
    _MOVE2269_OUT : ANY;
    _MOVE2282_ENO : BOOL;
    _MOVE2282_OUT : ANY;
    _MOVE2295_ENO : BOOL;
    _MOVE2295_OUT : ANY;
    _MOVE2308_ENO : BOOL;
    _MOVE2308_OUT : ANY;
    _MOVE2321_ENO : BOOL;
    _MOVE2321_OUT : ANY;
    _MOVE2334_ENO : BOOL;
    _MOVE2334_OUT : ANY;
  END_VAR

(* CFC diagram, written out as Structured Text *)
(* KNX Sending interval *)
(* KNX Master *)
Interval(IN := Interval.Q);
_ADD9_OUT := BOOL_TO_INT(Interval.Q) + i;
i := _ADD9_OUT;
_GT15_OUT := i > 77;
_MOVE19_OUT := MOVE(EN := _GT15_OUT, IN := 0, ENO => _MOVE19_ENO);
IF _MOVE19_ENO THEN i := _MOVE19_OUT; END_IF;
KNX_master_1(I_Port := IoConfig_Globals.KNX_EIB_TP1_Interface, bPortKNX := 1);
STLV59_563.STLV59_A_563_KNX_Card_1_Status := KNX_master_1.sStatus = 'OK';
(* Rom 001 *)
(* RB601_V *)
(* RB601_HVAC *)
M1_001_001_RB601_V(bPortKNX := 1, dwIndex_DPT := 1, typDPT := typDPT);
_MOVE46_OUT := MOVE(EN := M1_001_001_RB601_V.xUpdate_PLC, IN := M1_001_001_RB601_V.xSwitch_OUT, ENO => _MOVE46_ENO);
IF _MOVE46_ENO THEN STLV59_563.STLV59_A_563_001.RB601_V := _MOVE46_OUT; END_IF;
M1_002_001_RB601_HVAC(bPortKNX := 1, dwIndex_DPT := 2, typDPT := typDPT);
_MOVE59_OUT := MOVE(EN := M1_002_001_RB601_HVAC.xUpdate_PLC, IN := M1_002_001_RB601_HVAC.xSwitch_OUT, ENO => _MOVE59_ENO);
IF _MOVE59_ENO THEN STLV59_563.STLV59_A_563_001.RB601_HVAC := _MOVE59_OUT; END_IF;
(* RT601_CT *)
(* RY601_CV *)
M1_003_001_RT601_CT(bPortKNX := 1, dwIndex_DPT := 3, typDPT := typDPT);
_MOVE72_OUT := MOVE(EN := M1_003_001_RT601_CT.xUpdate_PLC, IN := M1_003_001_RT601_CT.rValue_OUT, ENO => _MOVE72_ENO);
IF _MOVE72_ENO THEN STLV59_563.STLV59_A_563_001.RT601_CT := _MOVE72_OUT; END_IF;
M1_004_001_RY601_CV(bPortKNX := 1, dwIndex_DPT := 4, typDPT := typDPT);
_MOVE85_OUT := MOVE(EN := M1_004_001_RY601_CV.xUpdate_PLC, IN := M1_004_001_RY601_CV.rValue_OUT, ENO => _MOVE85_ENO);
IF _MOVE85_ENO THEN STLV59_563.STLV59_A_563_001.RY601_CV := _MOVE85_OUT; END_IF;
(* LH601_OP *)
(* LH601_CMD *)
M1_005_001_LH601_OP(bPortKNX := 1, dwIndex_DPT := 5, rValue_IN := STLV59_563.STLV59_A_563_001.LH601_OP, xUpdate_KNX := i = 0, typDPT := typDPT);
M1_006_001_LH601_CMD(bPortKNX := 1, dwIndex_DPT := 6, xSwitch_IN := STLV59_563.STLV59_A_563_001.LH601_CMD, xUpdate_KNX := i = 1, typDPT := typDPT);
(* LC601_OP *)
(* LC601_CMD *)
M1_007_001_LC601_OP(bPortKNX := 1, dwIndex_DPT := 7, rValue_IN := STLV59_563.STLV59_A_563_001.LC601_OP, xUpdate_KNX := i = 2, typDPT := typDPT);
M1_008_001_LC601_CMD(bPortKNX := 1, dwIndex_DPT := 8, xSwitch_IN := STLV59_563.STLV59_A_563_001.LC601_CMD, xUpdate_KNX := i = 3, typDPT := typDPT);
(* RT601_SP *)
(* RT601_SP Feedback *)
M1_009_001_RT601_SP(bPortKNX := 1, dwIndex_DPT := 9, rValue_IN := STLV59_563.STLV59_A_563_001.RT601_SP_D, xUpdate_KNX := NOT STLV59_563.STLV59_A_563_001.RB601_HVAC, typDPT := typDPT);
M1_010_001_RT601_SP_FB(bPortKNX := 1, dwIndex_DPT := 10, typDPT := typDPT);
_MOVE174_OUT := MOVE(EN := M1_010_001_RT601_SP_FB.xUpdate_PLC, IN := M1_010_001_RT601_SP_FB.rValue_OUT, ENO => _MOVE174_ENO);
IF _MOVE174_ENO THEN STLV59_563.STLV59_A_563_001.RT601_SP_IN := _MOVE174_OUT; END_IF;
(* LU601_V *)
(* LU601_AL *)
M1_011_001_LU601_V(bPortKNX := 1, dwIndex_DPT := 11, typDPT := typDPT);
_MOVE187_OUT := MOVE(EN := M1_011_001_LU601_V.xUpdate_PLC, IN := M1_011_001_LU601_V.xSwitch_OUT, ENO => _MOVE187_ENO);
IF _MOVE187_ENO THEN STLV59_563.STLV59_A_563_001.LU601_V := _MOVE187_OUT; END_IF;
M1_012_001_LU601_AL(bPortKNX := 1, dwIndex_DPT := 12, typDPT := typDPT);
_MOVE200_OUT := MOVE(EN := M1_012_001_LU601_AL.xUpdate_PLC, IN := M1_012_001_LU601_AL.xSwitch_OUT, ENO => _MOVE200_ENO);
IF _MOVE200_ENO THEN STLV59_563.STLV59_A_563_001.LU601_AL := _MOVE200_OUT; END_IF;
(* LU601_CMD *)
(* OPM_001 *)
M1_013_001_LU601_CMD(bPortKNX := 1, dwIndex_DPT := 13, xSwitch_IN := STLV59_563.STLV59_A_563_001.LU601_CMD, xUpdate_KNX := i = 4, typDPT := typDPT);
M1_014_001_OPM_001(bPortKNX := 1, dwIndex_DPT := 14, bIN := STLV59_563.STLV59_A_563_001.OPM_001, xUpdate_KNX := i = 5, typDPT := typDPT);
(* Rom 002 *)
(* RB601_V *)
(* RB602_V *)
M1_015_002_RB601_V(bPortKNX := 1, dwIndex_DPT := 15, typDPT := typDPT);
_MOVE246_OUT := MOVE(EN := M1_015_002_RB601_V.xUpdate_PLC, IN := M1_015_002_RB601_V.xSwitch_OUT, ENO => _MOVE246_ENO);
IF _MOVE246_ENO THEN STLV59_563.STLV59_A_563_002.RB601_V := _MOVE246_OUT; END_IF;
M1_016_002_RB602_V(bPortKNX := 1, dwIndex_DPT := 16, typDPT := typDPT);
_MOVE259_OUT := MOVE(EN := M1_016_002_RB602_V.xUpdate_PLC, IN := M1_016_002_RB602_V.xSwitch_OUT, ENO => _MOVE259_ENO);
IF _MOVE259_ENO THEN STLV59_563.STLV59_A_563_002.RB602_V := _MOVE259_OUT; END_IF;
(* RB603_V *)
(* RB601_HVAC *)
M1_017_002_RB603_V(bPortKNX := 1, dwIndex_DPT := 17, typDPT := typDPT);
_MOVE272_OUT := MOVE(EN := M1_017_002_RB603_V.xUpdate_PLC, IN := M1_017_002_RB603_V.xSwitch_OUT, ENO => _MOVE272_ENO);
IF _MOVE272_ENO THEN STLV59_563.STLV59_A_563_002.RB603_V := _MOVE272_OUT; END_IF;
M1_018_002_RB601_HVAC(bPortKNX := 1, dwIndex_DPT := 18, typDPT := typDPT);
_MOVE285_OUT := MOVE(EN := M1_018_002_RB601_HVAC.xUpdate_PLC, IN := M1_018_002_RB601_HVAC.xSwitch_OUT, ENO => _MOVE285_ENO);
IF _MOVE285_ENO THEN STLV59_563.STLV59_A_563_002.RB601_HVAC := _MOVE285_OUT; END_IF;
(* RB602_HVAC *)
(* RB603_HVAC *)
M1_019_002_RB602_HVAC(bPortKNX := 1, dwIndex_DPT := 19, typDPT := typDPT);
_MOVE298_OUT := MOVE(EN := M1_019_002_RB602_HVAC.xUpdate_PLC, IN := M1_019_002_RB602_HVAC.xSwitch_OUT, ENO => _MOVE298_ENO);
IF _MOVE298_ENO THEN STLV59_563.STLV59_A_563_002.RB602_HVAC := _MOVE298_OUT; END_IF;
M1_020_002_RB603_HVAC(bPortKNX := 1, dwIndex_DPT := 20, typDPT := typDPT);
_MOVE311_OUT := MOVE(EN := M1_020_002_RB603_HVAC.xUpdate_PLC, IN := M1_020_002_RB603_HVAC.xSwitch_OUT, ENO => _MOVE311_ENO);
IF _MOVE311_ENO THEN STLV59_563.STLV59_A_563_002.RB603_HVAC := _MOVE311_OUT; END_IF;
(* RT601_CT *)
(* RT602_CT *)
M1_021_002_RT601_CT(bPortKNX := 1, dwIndex_DPT := 21, typDPT := typDPT);
_MOVE324_OUT := MOVE(EN := M1_021_002_RT601_CT.xUpdate_PLC, IN := M1_021_002_RT601_CT.rValue_OUT, ENO => _MOVE324_ENO);
IF _MOVE324_ENO THEN STLV59_563.STLV59_A_563_002.RT601_CT := _MOVE324_OUT; END_IF;
M1_022_002_RT602_CT(bPortKNX := 1, dwIndex_DPT := 22, typDPT := typDPT);
_MOVE337_OUT := MOVE(EN := M1_022_002_RT602_CT.xUpdate_PLC, IN := M1_022_002_RT602_CT.rValue_OUT, ENO => _MOVE337_ENO);
IF _MOVE337_ENO THEN STLV59_563.STLV59_A_563_002.RT602_CT := _MOVE337_OUT; END_IF;
(* RT603_CT *)
(* RY601_CV *)
M1_023_002_RT603_CT(bPortKNX := 1, dwIndex_DPT := 23, typDPT := typDPT);
_MOVE350_OUT := MOVE(EN := M1_023_002_RT603_CT.xUpdate_PLC, IN := M1_023_002_RT603_CT.rValue_OUT, ENO => _MOVE350_ENO);
IF _MOVE350_ENO THEN STLV59_563.STLV59_A_563_002.RT603_CT := _MOVE350_OUT; END_IF;
M1_024_002_RY601_CV(bPortKNX := 1, dwIndex_DPT := 24, typDPT := typDPT);
_MOVE363_OUT := MOVE(EN := M1_024_002_RY601_CV.xUpdate_PLC, IN := M1_024_002_RY601_CV.rValue_OUT, ENO => _MOVE363_ENO);
IF _MOVE363_ENO THEN STLV59_563.STLV59_A_563_002.RY601_CV := _MOVE363_OUT; END_IF;
(* RY602_CV *)
(* RY603_CV *)
M1_025_002_RY602_CV(bPortKNX := 1, dwIndex_DPT := 25, typDPT := typDPT);
_MOVE376_OUT := MOVE(EN := M1_025_002_RY602_CV.xUpdate_PLC, IN := M1_025_002_RY602_CV.rValue_OUT, ENO => _MOVE376_ENO);
IF _MOVE376_ENO THEN STLV59_563.STLV59_A_563_002.RY602_CV := _MOVE376_OUT; END_IF;
M1_026_002_RY603_CV(bPortKNX := 1, dwIndex_DPT := 26, typDPT := typDPT);
_MOVE389_OUT := MOVE(EN := M1_026_002_RY603_CV.xUpdate_PLC, IN := M1_026_002_RY603_CV.rValue_OUT, ENO => _MOVE389_ENO);
IF _MOVE389_ENO THEN STLV59_563.STLV59_A_563_002.RY603_CV := _MOVE389_OUT; END_IF;
(* LH601_OP *)
(* LH602_OP *)
M1_027_002_LH601_OP(bPortKNX := 1, dwIndex_DPT := 27, rValue_IN := STLV59_563.STLV59_A_563_002.LH601_OP, xUpdate_KNX := i = 6, typDPT := typDPT);
M1_028_002_LH602_OP(bPortKNX := 1, dwIndex_DPT := 28, rValue_IN := STLV59_563.STLV59_A_563_002.LH602_OP, xUpdate_KNX := i = 7, typDPT := typDPT);
(* LH603_OP *)
(* LH601_CMD *)
M1_029_002_LH603_OP(bPortKNX := 1, dwIndex_DPT := 29, rValue_IN := STLV59_563.STLV59_A_563_002.LH603_OP, xUpdate_KNX := i = 8, typDPT := typDPT);
M1_030_002_LH601_CMD(bPortKNX := 1, dwIndex_DPT := 30, xSwitch_IN := STLV59_563.STLV59_A_563_002.LH601_CMD, xUpdate_KNX := i = 9, typDPT := typDPT);
(* LH602_CMD *)
(* LH603_CMD *)
M1_031_002_LH602_CMD(bPortKNX := 1, dwIndex_DPT := 31, xSwitch_IN := STLV59_563.STLV59_A_563_002.LH602_CMD, xUpdate_KNX := i = 10, typDPT := typDPT);
M1_032_002_LH603_CMD(bPortKNX := 1, dwIndex_DPT := 32, xSwitch_IN := STLV59_563.STLV59_A_563_002.LH603_CMD, xUpdate_KNX := i = 11, typDPT := typDPT);
(* LC601_OP *)
(* LC602_OP *)
M1_033_002_LC601_OP(bPortKNX := 1, dwIndex_DPT := 33, rValue_IN := STLV59_563.STLV59_A_563_002.LC601_OP, xUpdate_KNX := i = 12, typDPT := typDPT);
M1_034_002_LC602_OP(bPortKNX := 1, dwIndex_DPT := 34, rValue_IN := STLV59_563.STLV59_A_563_002.LC602_OP, xUpdate_KNX := i = 13, typDPT := typDPT);
(* LC603_OP *)
(* LC601_CMD *)
M1_035_002_LC603_OP(bPortKNX := 1, dwIndex_DPT := 35, rValue_IN := STLV59_563.STLV59_A_563_002.LC603_OP, xUpdate_KNX := i = 14, typDPT := typDPT);
M1_036_002_LC601_CMD(bPortKNX := 1, dwIndex_DPT := 36, xSwitch_IN := STLV59_563.STLV59_A_563_002.LC601_CMD, xUpdate_KNX := i = 15, typDPT := typDPT);
(* LC602_CMD *)
(* LC603_CMD *)
M1_037_002_LC602_CMD(bPortKNX := 1, dwIndex_DPT := 37, xSwitch_IN := STLV59_563.STLV59_A_563_002.LC602_CMD, xUpdate_KNX := i = 16, typDPT := typDPT);
M1_038_002_LC603_CMD(bPortKNX := 1, dwIndex_DPT := 38, xSwitch_IN := STLV59_563.STLV59_A_563_002.LC603_CMD, xUpdate_KNX := i = 17, typDPT := typDPT);
(* RT601_SP *)
(* RT602_SP *)
M1_039_002_RT601_SP(bPortKNX := 1, dwIndex_DPT := 39, rValue_IN := STLV59_563.STLV59_A_563_002.RT601_SP_D, xUpdate_KNX := NOT STLV59_563.STLV59_A_563_002.RB601_HVAC, typDPT := typDPT);
M1_040_002_RT602_SP(bPortKNX := 1, dwIndex_DPT := 40, rValue_IN := STLV59_563.STLV59_A_563_002.RT602_SP, xUpdate_KNX := NOT STLV59_563.STLV59_A_563_002.RB601_HVAC, typDPT := typDPT);
(* RT603_SP *)
(* RT601_SP Feedback *)
M1_041_002_RT603_SP(bPortKNX := 1, dwIndex_DPT := 41, rValue_IN := STLV59_563.STLV59_A_563_002.RT603_SP, xUpdate_KNX := NOT STLV59_563.STLV59_A_563_002.RB601_HVAC, typDPT := typDPT);
M1_042_002_RT601_SP_FB(bPortKNX := 1, dwIndex_DPT := 42, typDPT := typDPT);
_MOVE630_OUT := MOVE(EN := M1_042_002_RT601_SP_FB.xUpdate_PLC, IN := M1_042_002_RT601_SP_FB.rValue_OUT, ENO => _MOVE630_ENO);
IF _MOVE630_ENO THEN STLV59_563.STLV59_A_563_002.RT601_SP_IN := _MOVE630_OUT; END_IF;
(* RT602_SP Feedback *)
(* RT603_SP Feedback *)
M1_043_002_RT602_SP_FB(bPortKNX := 1, dwIndex_DPT := 43, typDPT := typDPT);
_MOVE643_OUT := MOVE(EN := M1_043_002_RT602_SP_FB.xUpdate_PLC, IN := M1_043_002_RT602_SP_FB.rValue_OUT, ENO => _MOVE643_ENO);
IF _MOVE643_ENO THEN STLV59_563.STLV59_A_563_002.RT602_SP_IN := _MOVE643_OUT; END_IF;
M1_044_002_RT603_SP_FB(bPortKNX := 1, dwIndex_DPT := 44, typDPT := typDPT);
_MOVE656_OUT := MOVE(EN := M1_044_002_RT603_SP_FB.xUpdate_PLC, IN := M1_044_002_RT603_SP_FB.rValue_OUT, ENO => _MOVE656_ENO);
IF _MOVE656_ENO THEN STLV59_563.STLV59_A_563_002.RT603_SP_IN := _MOVE656_OUT; END_IF;
(* LU601_V *)
(* LU602_V *)
M1_045_002_LU601_V(bPortKNX := 1, dwIndex_DPT := 45, typDPT := typDPT);
_MOVE669_OUT := MOVE(EN := M1_045_002_LU601_V.xUpdate_PLC, IN := M1_045_002_LU601_V.xSwitch_OUT, ENO => _MOVE669_ENO);
IF _MOVE669_ENO THEN STLV59_563.STLV59_A_563_002.LU601_V := _MOVE669_OUT; END_IF;
M1_046_002_LU602_V(bPortKNX := 1, dwIndex_DPT := 46, typDPT := typDPT);
_MOVE682_OUT := MOVE(EN := M1_046_002_LU602_V.xUpdate_PLC, IN := M1_046_002_LU602_V.xSwitch_OUT, ENO => _MOVE682_ENO);
IF _MOVE682_ENO THEN STLV59_563.STLV59_A_563_002.LU602_V := _MOVE682_OUT; END_IF;
(* LU603_V *)
(* LU601_AL *)
M1_047_002_LU603_V(bPortKNX := 1, dwIndex_DPT := 47, typDPT := typDPT);
_MOVE695_OUT := MOVE(EN := M1_047_002_LU603_V.xUpdate_PLC, IN := M1_047_002_LU603_V.xSwitch_OUT, ENO => _MOVE695_ENO);
IF _MOVE695_ENO THEN STLV59_563.STLV59_A_563_002.LU603_V := _MOVE695_OUT; END_IF;
M1_048_002_LU601_AL(bPortKNX := 1, dwIndex_DPT := 48, typDPT := typDPT);
_MOVE708_OUT := MOVE(EN := M1_048_002_LU601_AL.xUpdate_PLC, IN := M1_048_002_LU601_AL.xSwitch_OUT, ENO => _MOVE708_ENO);
IF _MOVE708_ENO THEN STLV59_563.STLV59_A_563_002.LU601_AL := _MOVE708_OUT; END_IF;
(* LU602_AL *)
(* LU603_AL *)
M1_049_002_LU602_AL(bPortKNX := 1, dwIndex_DPT := 49, typDPT := typDPT);
_MOVE721_OUT := MOVE(EN := M1_049_002_LU602_AL.xUpdate_PLC, IN := M1_049_002_LU602_AL.xSwitch_OUT, ENO => _MOVE721_ENO);
IF _MOVE721_ENO THEN STLV59_563.STLV59_A_563_002.LU602_AL := _MOVE721_OUT; END_IF;
M1_050_002_LU603_AL(bPortKNX := 1, dwIndex_DPT := 50, typDPT := typDPT);
_MOVE734_OUT := MOVE(EN := M1_050_002_LU603_AL.xUpdate_PLC, IN := M1_050_002_LU603_AL.xSwitch_OUT, ENO => _MOVE734_ENO);
IF _MOVE734_ENO THEN STLV59_563.STLV59_A_563_002.LU603_AL := _MOVE734_OUT; END_IF;
(* LU601_CMD *)
(* LU602_CMD *)
M1_051_002_LU601_CMD(bPortKNX := 1, dwIndex_DPT := 51, xSwitch_IN := STLV59_563.STLV59_A_563_002.LU601_CMD, xUpdate_KNX := i = 18, typDPT := typDPT);
M1_052_002_LU602_CMD(bPortKNX := 1, dwIndex_DPT := 52, xSwitch_IN := STLV59_563.STLV59_A_563_002.LU602_CMD, xUpdate_KNX := i = 19, typDPT := typDPT);
(* LU603_CMD *)
(* OPM_001 *)
M1_053_002_LU603_CMD(bPortKNX := 1, dwIndex_DPT := 53, xSwitch_IN := STLV59_563.STLV59_A_563_002.LU603_CMD, xUpdate_KNX := i = 20, typDPT := typDPT);
M1_054_002_OPM_001(bPortKNX := 1, dwIndex_DPT := 54, bIN := STLV59_563.STLV59_A_563_002.OPM_001, xUpdate_KNX := i = 21, typDPT := typDPT);
(* OPM_002 *)
(* OPM_003 *)
M1_055_002_OPM_002(bPortKNX := 1, dwIndex_DPT := 55, bIN := STLV59_563.STLV59_A_563_002.OPM_002, xUpdate_KNX := i = 22, typDPT := typDPT);
M1_056_002_OPM_003(bPortKNX := 1, dwIndex_DPT := 56, bIN := STLV59_563.STLV59_A_563_002.OPM_003, xUpdate_KNX := i = 23, typDPT := typDPT);
(* Rom 003 *)
(* RB601_V *)
(* RB602_V *)
M1_057_003_RB601_V(bPortKNX := 1, dwIndex_DPT := 57, typDPT := typDPT);
_MOVE844_OUT := MOVE(EN := M1_057_003_RB601_V.xUpdate_PLC, IN := M1_057_003_RB601_V.xSwitch_OUT, ENO => _MOVE844_ENO);
IF _MOVE844_ENO THEN STLV59_563.STLV59_A_563_003.RB601_V := _MOVE844_OUT; END_IF;
M1_058_003_RB602_V(bPortKNX := 1, dwIndex_DPT := 58, typDPT := typDPT);
_MOVE857_OUT := MOVE(EN := M1_058_003_RB602_V.xUpdate_PLC, IN := M1_058_003_RB602_V.xSwitch_OUT, ENO => _MOVE857_ENO);
IF _MOVE857_ENO THEN STLV59_563.STLV59_A_563_003.RB602_V := _MOVE857_OUT; END_IF;
(* RB603_V *)
(* RB604_V *)
M1_059_003_RB603_V(bPortKNX := 1, dwIndex_DPT := 59, typDPT := typDPT);
_MOVE870_OUT := MOVE(EN := M1_059_003_RB603_V.xUpdate_PLC, IN := M1_059_003_RB603_V.xSwitch_OUT, ENO => _MOVE870_ENO);
IF _MOVE870_ENO THEN STLV59_563.STLV59_A_563_003.RB603_V := _MOVE870_OUT; END_IF;
M1_060_003_RB604_V(bPortKNX := 1, dwIndex_DPT := 60, typDPT := typDPT);
_MOVE883_OUT := MOVE(EN := M1_060_003_RB604_V.xUpdate_PLC, IN := M1_060_003_RB604_V.xSwitch_OUT, ENO => _MOVE883_ENO);
IF _MOVE883_ENO THEN STLV59_563.STLV59_A_563_003.RB604_V := _MOVE883_OUT; END_IF;
(* RB605_V *)
(* RB606_V *)
M1_061_003_RB605_V(bPortKNX := 1, dwIndex_DPT := 61, typDPT := typDPT);
_MOVE896_OUT := MOVE(EN := M1_061_003_RB605_V.xUpdate_PLC, IN := M1_061_003_RB605_V.xSwitch_OUT, ENO => _MOVE896_ENO);
IF _MOVE896_ENO THEN STLV59_563.STLV59_A_563_003.RB605_V := _MOVE896_OUT; END_IF;
M1_062_003_RB606_V(bPortKNX := 1, dwIndex_DPT := 62, typDPT := typDPT);
_MOVE909_OUT := MOVE(EN := M1_062_003_RB606_V.xUpdate_PLC, IN := M1_062_003_RB606_V.xSwitch_OUT, ENO => _MOVE909_ENO);
IF _MOVE909_ENO THEN STLV59_563.STLV59_A_563_003.RB606_V := _MOVE909_OUT; END_IF;
(* RB607_V *)
(* RB608_V *)
M1_063_003_RB607_V(bPortKNX := 1, dwIndex_DPT := 63, typDPT := typDPT);
_MOVE922_OUT := MOVE(EN := M1_063_003_RB607_V.xUpdate_PLC, IN := M1_063_003_RB607_V.xSwitch_OUT, ENO => _MOVE922_ENO);
IF _MOVE922_ENO THEN STLV59_563.STLV59_A_563_003.RB607_V := _MOVE922_OUT; END_IF;
M1_064_003_RB608_V(bPortKNX := 1, dwIndex_DPT := 64, typDPT := typDPT);
_MOVE935_OUT := MOVE(EN := M1_064_003_RB608_V.xUpdate_PLC, IN := M1_064_003_RB608_V.xSwitch_OUT, ENO => _MOVE935_ENO);
IF _MOVE935_ENO THEN STLV59_563.STLV59_A_563_003.RB608_V := _MOVE935_OUT; END_IF;
(* RB609_V *)
(* RB601_HVAC *)
M1_065_003_RB609_V(bPortKNX := 1, dwIndex_DPT := 65, typDPT := typDPT);
_MOVE948_OUT := MOVE(EN := M1_065_003_RB609_V.xUpdate_PLC, IN := M1_065_003_RB609_V.xSwitch_OUT, ENO => _MOVE948_ENO);
IF _MOVE948_ENO THEN STLV59_563.STLV59_A_563_003.RB609_V := _MOVE948_OUT; END_IF;
M1_066_003_RB601_HVAC(bPortKNX := 1, dwIndex_DPT := 66, typDPT := typDPT);
_MOVE961_OUT := MOVE(EN := M1_066_003_RB601_HVAC.xUpdate_PLC, IN := M1_066_003_RB601_HVAC.xSwitch_OUT, ENO => _MOVE961_ENO);
IF _MOVE961_ENO THEN STLV59_563.STLV59_A_563_003.RB601_HVAC := _MOVE961_OUT; END_IF;
(* RB602_HVAC *)
(* RB603_HVAC *)
M1_067_003_RB602_HVAC(bPortKNX := 1, dwIndex_DPT := 67, typDPT := typDPT);
_MOVE974_OUT := MOVE(EN := M1_067_003_RB602_HVAC.xUpdate_PLC, IN := M1_067_003_RB602_HVAC.xSwitch_OUT, ENO => _MOVE974_ENO);
IF _MOVE974_ENO THEN STLV59_563.STLV59_A_563_003.RB602_HVAC := _MOVE974_OUT; END_IF;
M1_068_003_RB603_HVAC(bPortKNX := 1, dwIndex_DPT := 68, typDPT := typDPT);
_MOVE987_OUT := MOVE(EN := M1_068_003_RB603_HVAC.xUpdate_PLC, IN := M1_068_003_RB603_HVAC.xSwitch_OUT, ENO => _MOVE987_ENO);
IF _MOVE987_ENO THEN STLV59_563.STLV59_A_563_003.RB603_HVAC := _MOVE987_OUT; END_IF;
(* RB604_HVAC *)
(* RB605_HVAC *)
M1_069_003_RB604_HVAC(bPortKNX := 1, dwIndex_DPT := 69, typDPT := typDPT);
_MOVE1000_OUT := MOVE(EN := M1_069_003_RB604_HVAC.xUpdate_PLC, IN := M1_069_003_RB604_HVAC.xSwitch_OUT, ENO => _MOVE1000_ENO);
IF _MOVE1000_ENO THEN STLV59_563.STLV59_A_563_003.RB604_HVAC := _MOVE1000_OUT; END_IF;
M1_070_003_RB605_HVAC(bPortKNX := 1, dwIndex_DPT := 70, typDPT := typDPT);
_MOVE1013_OUT := MOVE(EN := M1_070_003_RB605_HVAC.xUpdate_PLC, IN := M1_070_003_RB605_HVAC.xSwitch_OUT, ENO => _MOVE1013_ENO);
IF _MOVE1013_ENO THEN STLV59_563.STLV59_A_563_003.RB605_HVAC := _MOVE1013_OUT; END_IF;
(* RB606_HVAC *)
(* RB607_HVAC *)
M1_071_003_RB606_HVAC(bPortKNX := 1, dwIndex_DPT := 71, typDPT := typDPT);
_MOVE1026_OUT := MOVE(EN := M1_071_003_RB606_HVAC.xUpdate_PLC, IN := M1_071_003_RB606_HVAC.xSwitch_OUT, ENO => _MOVE1026_ENO);
IF _MOVE1026_ENO THEN STLV59_563.STLV59_A_563_003.RB606_HVAC := _MOVE1026_OUT; END_IF;
M1_072_003_RB607_HVAC(bPortKNX := 1, dwIndex_DPT := 72, typDPT := typDPT);
_MOVE1039_OUT := MOVE(EN := M1_072_003_RB607_HVAC.xUpdate_PLC, IN := M1_072_003_RB607_HVAC.xSwitch_OUT, ENO => _MOVE1039_ENO);
IF _MOVE1039_ENO THEN STLV59_563.STLV59_A_563_003.RB607_HVAC := _MOVE1039_OUT; END_IF;
(* RB608_HVAC *)
(* RB609_HVAC *)
M1_073_003_RB608_HVAC(bPortKNX := 1, dwIndex_DPT := 73, typDPT := typDPT);
_MOVE1052_OUT := MOVE(EN := M1_073_003_RB608_HVAC.xUpdate_PLC, IN := M1_073_003_RB608_HVAC.xSwitch_OUT, ENO => _MOVE1052_ENO);
IF _MOVE1052_ENO THEN STLV59_563.STLV59_A_563_003.RB608_HVAC := _MOVE1052_OUT; END_IF;
M1_074_003_RB609_HVAC(bPortKNX := 1, dwIndex_DPT := 74, typDPT := typDPT);
_MOVE1065_OUT := MOVE(EN := M1_074_003_RB609_HVAC.xUpdate_PLC, IN := M1_074_003_RB609_HVAC.xSwitch_OUT, ENO => _MOVE1065_ENO);
IF _MOVE1065_ENO THEN STLV59_563.STLV59_A_563_003.RB609_HVAC := _MOVE1065_OUT; END_IF;
(* RT601_CT *)
(* RT602_CT *)
M1_075_003_RT601_CT(bPortKNX := 1, dwIndex_DPT := 75, typDPT := typDPT);
_MOVE1078_OUT := MOVE(EN := M1_075_003_RT601_CT.xUpdate_PLC, IN := M1_075_003_RT601_CT.rValue_OUT, ENO => _MOVE1078_ENO);
IF _MOVE1078_ENO THEN STLV59_563.STLV59_A_563_003.RT601_CT := _MOVE1078_OUT; END_IF;
M1_076_003_RT602_CT(bPortKNX := 1, dwIndex_DPT := 76, typDPT := typDPT);
_MOVE1091_OUT := MOVE(EN := M1_076_003_RT602_CT.xUpdate_PLC, IN := M1_076_003_RT602_CT.rValue_OUT, ENO => _MOVE1091_ENO);
IF _MOVE1091_ENO THEN STLV59_563.STLV59_A_563_003.RT602_CT := _MOVE1091_OUT; END_IF;
(* RT603_CT *)
(* RT604_CT *)
M1_077_003_RT603_CT(bPortKNX := 1, dwIndex_DPT := 77, typDPT := typDPT);
_MOVE1104_OUT := MOVE(EN := M1_077_003_RT603_CT.xUpdate_PLC, IN := M1_077_003_RT603_CT.rValue_OUT, ENO => _MOVE1104_ENO);
IF _MOVE1104_ENO THEN STLV59_563.STLV59_A_563_003.RT603_CT := _MOVE1104_OUT; END_IF;
M1_078_003_RT604_CT(bPortKNX := 1, dwIndex_DPT := 78, typDPT := typDPT);
_MOVE1117_OUT := MOVE(EN := M1_078_003_RT604_CT.xUpdate_PLC, IN := M1_078_003_RT604_CT.rValue_OUT, ENO => _MOVE1117_ENO);
IF _MOVE1117_ENO THEN STLV59_563.STLV59_A_563_003.RT604_CT := _MOVE1117_OUT; END_IF;
(* RT605_CT *)
(* RT606_CT *)
M1_079_003_RT605_CT(bPortKNX := 1, dwIndex_DPT := 79, typDPT := typDPT);
_MOVE1130_OUT := MOVE(EN := M1_079_003_RT605_CT.xUpdate_PLC, IN := M1_079_003_RT605_CT.rValue_OUT, ENO => _MOVE1130_ENO);
IF _MOVE1130_ENO THEN STLV59_563.STLV59_A_563_003.RT605_CT := _MOVE1130_OUT; END_IF;
M1_080_003_RT606_CT(bPortKNX := 1, dwIndex_DPT := 80, typDPT := typDPT);
_MOVE1143_OUT := MOVE(EN := M1_080_003_RT606_CT.xUpdate_PLC, IN := M1_080_003_RT606_CT.rValue_OUT, ENO => _MOVE1143_ENO);
IF _MOVE1143_ENO THEN STLV59_563.STLV59_A_563_003.RT606_CT := _MOVE1143_OUT; END_IF;
(* RT607_CT *)
(* RT608_CT *)
M1_081_003_RT607_CT(bPortKNX := 1, dwIndex_DPT := 81, typDPT := typDPT);
_MOVE1156_OUT := MOVE(EN := M1_081_003_RT607_CT.xUpdate_PLC, IN := M1_081_003_RT607_CT.rValue_OUT, ENO => _MOVE1156_ENO);
IF _MOVE1156_ENO THEN STLV59_563.STLV59_A_563_003.RT607_CT := _MOVE1156_OUT; END_IF;
M1_082_003_RT608_CT(bPortKNX := 1, dwIndex_DPT := 82, typDPT := typDPT);
_MOVE1169_OUT := MOVE(EN := M1_082_003_RT608_CT.xUpdate_PLC, IN := M1_082_003_RT608_CT.rValue_OUT, ENO => _MOVE1169_ENO);
IF _MOVE1169_ENO THEN STLV59_563.STLV59_A_563_003.RT608_CT := _MOVE1169_OUT; END_IF;
(* RT609_CT *)
(* RY601_CV *)
M1_083_003_RT609_CT(bPortKNX := 1, dwIndex_DPT := 83, typDPT := typDPT);
_MOVE1182_OUT := MOVE(EN := M1_083_003_RT609_CT.xUpdate_PLC, IN := M1_083_003_RT609_CT.rValue_OUT, ENO => _MOVE1182_ENO);
IF _MOVE1182_ENO THEN STLV59_563.STLV59_A_563_003.RT609_CT := _MOVE1182_OUT; END_IF;
M1_084_003_RY601_CV(bPortKNX := 1, dwIndex_DPT := 84, typDPT := typDPT);
_MOVE1195_OUT := MOVE(EN := M1_084_003_RY601_CV.xUpdate_PLC, IN := M1_084_003_RY601_CV.rValue_OUT, ENO => _MOVE1195_ENO);
IF _MOVE1195_ENO THEN STLV59_563.STLV59_A_563_003.RY601_CV := _MOVE1195_OUT; END_IF;
(* RY602_CV *)
(* RY603_CV *)
M1_085_003_RY602_CV(bPortKNX := 1, dwIndex_DPT := 85, typDPT := typDPT);
_MOVE1208_OUT := MOVE(EN := M1_085_003_RY602_CV.xUpdate_PLC, IN := M1_085_003_RY602_CV.rValue_OUT, ENO => _MOVE1208_ENO);
IF _MOVE1208_ENO THEN STLV59_563.STLV59_A_563_003.RY602_CV := _MOVE1208_OUT; END_IF;
M1_086_003_RY603_CV(bPortKNX := 1, dwIndex_DPT := 86, typDPT := typDPT);
_MOVE1221_OUT := MOVE(EN := M1_086_003_RY603_CV.xUpdate_PLC, IN := M1_086_003_RY603_CV.rValue_OUT, ENO => _MOVE1221_ENO);
IF _MOVE1221_ENO THEN STLV59_563.STLV59_A_563_003.RY603_CV := _MOVE1221_OUT; END_IF;
(* RY604_CV *)
(* RY605_CV *)
M1_087_003_RY604_CV(bPortKNX := 1, dwIndex_DPT := 87, typDPT := typDPT);
_MOVE1234_OUT := MOVE(EN := M1_087_003_RY604_CV.xUpdate_PLC, IN := M1_087_003_RY604_CV.rValue_OUT, ENO => _MOVE1234_ENO);
IF _MOVE1234_ENO THEN STLV59_563.STLV59_A_563_003.RY604_CV := _MOVE1234_OUT; END_IF;
M1_088_003_RY605_CV(bPortKNX := 1, dwIndex_DPT := 88, typDPT := typDPT);
_MOVE1247_OUT := MOVE(EN := M1_088_003_RY605_CV.xUpdate_PLC, IN := M1_088_003_RY605_CV.rValue_OUT, ENO => _MOVE1247_ENO);
IF _MOVE1247_ENO THEN STLV59_563.STLV59_A_563_003.RY605_CV := _MOVE1247_OUT; END_IF;
(* RY606_CV *)
(* RY607_CV *)
M1_089_003_RY606_CV(bPortKNX := 1, dwIndex_DPT := 89, typDPT := typDPT);
_MOVE1260_OUT := MOVE(EN := M1_089_003_RY606_CV.xUpdate_PLC, IN := M1_089_003_RY606_CV.rValue_OUT, ENO => _MOVE1260_ENO);
IF _MOVE1260_ENO THEN STLV59_563.STLV59_A_563_003.RY606_CV := _MOVE1260_OUT; END_IF;
M1_090_003_RY607_CV(bPortKNX := 1, dwIndex_DPT := 90, typDPT := typDPT);
_MOVE1273_OUT := MOVE(EN := M1_090_003_RY607_CV.xUpdate_PLC, IN := M1_090_003_RY607_CV.rValue_OUT, ENO => _MOVE1273_ENO);
IF _MOVE1273_ENO THEN STLV59_563.STLV59_A_563_003.RY607_CV := _MOVE1273_OUT; END_IF;
(* RY608_CV *)
(* RY609_CV *)
M1_091_003_RY608_CV(bPortKNX := 1, dwIndex_DPT := 91, typDPT := typDPT);
_MOVE1286_OUT := MOVE(EN := M1_091_003_RY608_CV.xUpdate_PLC, IN := M1_091_003_RY608_CV.rValue_OUT, ENO => _MOVE1286_ENO);
IF _MOVE1286_ENO THEN STLV59_563.STLV59_A_563_003.RY608_CV := _MOVE1286_OUT; END_IF;
M1_092_003_RY609_CV(bPortKNX := 1, dwIndex_DPT := 92, typDPT := typDPT);
_MOVE1299_OUT := MOVE(EN := M1_092_003_RY609_CV.xUpdate_PLC, IN := M1_092_003_RY609_CV.rValue_OUT, ENO => _MOVE1299_ENO);
IF _MOVE1299_ENO THEN STLV59_563.STLV59_A_563_003.RY609_CV := _MOVE1299_OUT; END_IF;
(* LH601_OP *)
(* LH602_OP *)
M1_093_003_LH601_OP(bPortKNX := 1, dwIndex_DPT := 93, rValue_IN := STLV59_563.STLV59_A_563_003.LH601_OP, xUpdate_KNX := i = 24, typDPT := typDPT);
M1_094_003_LH602_OP(bPortKNX := 1, dwIndex_DPT := 94, rValue_IN := STLV59_563.STLV59_A_563_003.LH602_OP, xUpdate_KNX := i = 25, typDPT := typDPT);
(* LH603_OP *)
(* LH604_OP *)
M1_095_003_LH603_OP(bPortKNX := 1, dwIndex_DPT := 95, rValue_IN := STLV59_563.STLV59_A_563_003.LH603_OP, xUpdate_KNX := i = 26, typDPT := typDPT);
M1_096_003_LH604_OP(bPortKNX := 1, dwIndex_DPT := 96, rValue_IN := STLV59_563.STLV59_A_563_003.LH604_OP, xUpdate_KNX := i = 27, typDPT := typDPT);
(* LH605_OP *)
(* LH606_OP *)
M1_097_003_LH605_OP(bPortKNX := 1, dwIndex_DPT := 97, rValue_IN := STLV59_563.STLV59_A_563_003.LH605_OP, xUpdate_KNX := i = 28, typDPT := typDPT);
M1_098_003_LH606_OP(bPortKNX := 1, dwIndex_DPT := 98, rValue_IN := STLV59_563.STLV59_A_563_003.LH606_OP, xUpdate_KNX := i = 29, typDPT := typDPT);
(* LH607_OP *)
(* LH608_OP *)
M1_099_003_LH607_OP(bPortKNX := 1, dwIndex_DPT := 99, rValue_IN := STLV59_563.STLV59_A_563_003.LH607_OP, xUpdate_KNX := i = 30, typDPT := typDPT);
M1_0100_003_LH608_OP(bPortKNX := 1, dwIndex_DPT := 100, rValue_IN := STLV59_563.STLV59_A_563_003.LH608_OP, xUpdate_KNX := i = 31, typDPT := typDPT);
(* LH609_OP *)
(* LH601_CMD *)
M1_0101_003_LH609_OP(bPortKNX := 1, dwIndex_DPT := 101, rValue_IN := STLV59_563.STLV59_A_563_003.LH609_OP, xUpdate_KNX := i = 32, typDPT := typDPT);
M1_102_003_LH601_CMD(bPortKNX := 1, dwIndex_DPT := 102, xSwitch_IN := STLV59_563.STLV59_A_563_003.LH601_CMD, xUpdate_KNX := i = 33, typDPT := typDPT);
(* LH602_CMD *)
(* LH603_CMD *)
M1_103_003_LH602_CMD(bPortKNX := 1, dwIndex_DPT := 103, xSwitch_IN := STLV59_563.STLV59_A_563_003.LH602_CMD, xUpdate_KNX := i = 34, typDPT := typDPT);
M1_104_003_LH603_CMD(bPortKNX := 1, dwIndex_DPT := 104, xSwitch_IN := STLV59_563.STLV59_A_563_003.LH603_CMD, xUpdate_KNX := i = 35, typDPT := typDPT);
(* LH604_CMD *)
(* LH605_CMD *)
M1_105_003_LH604_CMD(bPortKNX := 1, dwIndex_DPT := 105, xSwitch_IN := STLV59_563.STLV59_A_563_003.LH604_CMD, xUpdate_KNX := i = 36, typDPT := typDPT);
M1_106_003_LH605_CMD(bPortKNX := 1, dwIndex_DPT := 106, xSwitch_IN := STLV59_563.STLV59_A_563_003.LH605_CMD, xUpdate_KNX := i = 37, typDPT := typDPT);
(* LH606_CMD *)
(* LH607_CMD *)
M1_107_003_LH606_CMD(bPortKNX := 1, dwIndex_DPT := 107, xSwitch_IN := STLV59_563.STLV59_A_563_003.LH606_CMD, xUpdate_KNX := i = 38, typDPT := typDPT);
M1_108_003_LH607_CMD(bPortKNX := 1, dwIndex_DPT := 108, xSwitch_IN := STLV59_563.STLV59_A_563_003.LH607_CMD, xUpdate_KNX := i = 39, typDPT := typDPT);
(* LH608_CMD *)
(* LH609_CMD *)
M1_109_003_LH608_CMD(bPortKNX := 1, dwIndex_DPT := 109, xSwitch_IN := STLV59_563.STLV59_A_563_003.LH608_CMD, xUpdate_KNX := i = 40, typDPT := typDPT);
M1_110_003_LH609_CMD(bPortKNX := 1, dwIndex_DPT := 110, xSwitch_IN := STLV59_563.STLV59_A_563_003.LH609_CMD, xUpdate_KNX := i = 41, typDPT := typDPT);
(* LC601_OP *)
(* LC602_OP *)
M1_111_003_LC601_OP(bPortKNX := 1, dwIndex_DPT := 111, rValue_IN := STLV59_563.STLV59_A_563_003.LC601_OP, xUpdate_KNX := i = 42, typDPT := typDPT);
M1_112_003_LC602_OP(bPortKNX := 1, dwIndex_DPT := 112, rValue_IN := STLV59_563.STLV59_A_563_003.LC602_OP, xUpdate_KNX := i = 43, typDPT := typDPT);
(* LC603_OP *)
(* LC604_OP *)
M1_113_003_LC603_OP(bPortKNX := 1, dwIndex_DPT := 113, rValue_IN := STLV59_563.STLV59_A_563_003.LC603_OP, xUpdate_KNX := i = 44, typDPT := typDPT);
M1_114_003_LC604_OP(bPortKNX := 1, dwIndex_DPT := 114, rValue_IN := STLV59_563.STLV59_A_563_003.LC604_OP, xUpdate_KNX := i = 45, typDPT := typDPT);
(* LC605_OP *)
(* LC606_OP *)
M1_115_003_LC605_OP(bPortKNX := 1, dwIndex_DPT := 115, rValue_IN := STLV59_563.STLV59_A_563_003.LC605_OP, xUpdate_KNX := i = 46, typDPT := typDPT);
M1_116_003_LC606_OP(bPortKNX := 1, dwIndex_DPT := 116, rValue_IN := STLV59_563.STLV59_A_563_003.LC606_OP, xUpdate_KNX := i = 47, typDPT := typDPT);
(* LC607_OP *)
(* LC608_OP *)
M1_117_003_LC607_OP(bPortKNX := 1, dwIndex_DPT := 117, rValue_IN := STLV59_563.STLV59_A_563_003.LC607_OP, xUpdate_KNX := i = 48, typDPT := typDPT);
M1_118_003_LC608_OP(bPortKNX := 1, dwIndex_DPT := 118, rValue_IN := STLV59_563.STLV59_A_563_003.LC608_OP, xUpdate_KNX := i = 49, typDPT := typDPT);
(* LC609_OP *)
(* LC601_CMD *)
M1_119_003_LC609_OP(bPortKNX := 1, dwIndex_DPT := 119, rValue_IN := STLV59_563.STLV59_A_563_003.LC609_OP, xUpdate_KNX := i = 50, typDPT := typDPT);
M1_120_003_LC601_CMD(bPortKNX := 1, dwIndex_DPT := 120, xSwitch_IN := STLV59_563.STLV59_A_563_003.LC601_CMD, xUpdate_KNX := i = 51, typDPT := typDPT);
(* LC602_CMD *)
(* LC603_CMD *)
M1_121_003_LC602_CMD(bPortKNX := 1, dwIndex_DPT := 121, xSwitch_IN := STLV59_563.STLV59_A_563_003.LC602_CMD, xUpdate_KNX := i = 52, typDPT := typDPT);
M1_122_003_LC603_CMD(bPortKNX := 1, dwIndex_DPT := 122, xSwitch_IN := STLV59_563.STLV59_A_563_003.LC603_CMD, xUpdate_KNX := i = 53, typDPT := typDPT);
(* LC604_CMD *)
(* LC605_CMD *)
M1_123_003_LC604_CMD(bPortKNX := 1, dwIndex_DPT := 123, xSwitch_IN := STLV59_563.STLV59_A_563_003.LC604_CMD, xUpdate_KNX := i = 54, typDPT := typDPT);
M1_124_003_LC605_CMD(bPortKNX := 1, dwIndex_DPT := 124, xSwitch_IN := STLV59_563.STLV59_A_563_003.LC605_CMD, xUpdate_KNX := i = 55, typDPT := typDPT);
(* LC606_CMD *)
(* LC607_CMD *)
M1_125_003_LC606_CMD(bPortKNX := 1, dwIndex_DPT := 125, xSwitch_IN := STLV59_563.STLV59_A_563_003.LC606_CMD, xUpdate_KNX := i = 56, typDPT := typDPT);
M1_126_003_LC607_CMD(bPortKNX := 1, dwIndex_DPT := 126, xSwitch_IN := STLV59_563.STLV59_A_563_003.LC607_CMD, xUpdate_KNX := i = 57, typDPT := typDPT);
(* LC608_CMD *)
(* LC609_CMD *)
M1_127_003_LC608_CMD(bPortKNX := 1, dwIndex_DPT := 127, xSwitch_IN := STLV59_563.STLV59_A_563_003.LC608_CMD, xUpdate_KNX := i = 58, typDPT := typDPT);
M1_128_003_LC609_CMD(bPortKNX := 1, dwIndex_DPT := 128, xSwitch_IN := STLV59_563.STLV59_A_563_003.LC609_CMD, xUpdate_KNX := i = 59, typDPT := typDPT);
(* RT601_SP *)
(* RT602_SP *)
M1_129_003_RT601_SP(bPortKNX := 1, dwIndex_DPT := 129, rValue_IN := STLV59_563.STLV59_A_563_003.RT601_SP_D, xUpdate_KNX := NOT STLV59_563.STLV59_A_563_003.RB601_HVAC, typDPT := typDPT);
M1_130_003_RT602_SP(bPortKNX := 1, dwIndex_DPT := 130, rValue_IN := STLV59_563.STLV59_A_563_003.RT602_SP, xUpdate_KNX := NOT STLV59_563.STLV59_A_563_003.RB601_HVAC, typDPT := typDPT);
(* RT603_SP *)
(* RT604_SP *)
M1_131_003_RT603_SP(bPortKNX := 1, dwIndex_DPT := 131, rValue_IN := STLV59_563.STLV59_A_563_003.RT603_SP, xUpdate_KNX := NOT STLV59_563.STLV59_A_563_003.RB601_HVAC, typDPT := typDPT);
M1_132_003_RT604_SP(bPortKNX := 1, dwIndex_DPT := 132, rValue_IN := STLV59_563.STLV59_A_563_003.RT604_SP, xUpdate_KNX := NOT STLV59_563.STLV59_A_563_003.RB601_HVAC, typDPT := typDPT);
(* RT605_SP *)
(* RT606_SP *)
M1_133_003_RT605_SP(bPortKNX := 1, dwIndex_DPT := 133, rValue_IN := STLV59_563.STLV59_A_563_003.RT605_SP, xUpdate_KNX := NOT STLV59_563.STLV59_A_563_003.RB601_HVAC, typDPT := typDPT);
M1_134_003_RT606_SP(bPortKNX := 1, dwIndex_DPT := 134, rValue_IN := STLV59_563.STLV59_A_563_003.RT606_SP, xUpdate_KNX := NOT STLV59_563.STLV59_A_563_003.RB601_HVAC, typDPT := typDPT);
(* RT607_SP *)
(* RT608_SP *)
M1_135_003_RT607_SP(bPortKNX := 1, dwIndex_DPT := 135, rValue_IN := STLV59_563.STLV59_A_563_003.RT607_SP, xUpdate_KNX := NOT STLV59_563.STLV59_A_563_003.RB601_HVAC, typDPT := typDPT);
M1_136_003_RT608_SP(bPortKNX := 1, dwIndex_DPT := 136, rValue_IN := STLV59_563.STLV59_A_563_003.RT608_SP, xUpdate_KNX := NOT STLV59_563.STLV59_A_563_003.RB601_HVAC, typDPT := typDPT);
(* RT609_SP *)
(* RT601_SP Feedback *)
M1_137_003_RT609_SP(bPortKNX := 1, dwIndex_DPT := 137, rValue_IN := STLV59_563.STLV59_A_563_003.RT609_SP, xUpdate_KNX := NOT STLV59_563.STLV59_A_563_003.RB601_HVAC, typDPT := typDPT);
M1_138_003_RT601_SP_FB(bPortKNX := 1, dwIndex_DPT := 138, typDPT := typDPT);
_MOVE1996_OUT := MOVE(EN := M1_138_003_RT601_SP_FB.xUpdate_PLC, IN := M1_138_003_RT601_SP_FB.rValue_OUT, ENO => _MOVE1996_ENO);
IF _MOVE1996_ENO THEN STLV59_563.STLV59_A_563_003.RT601_SP_IN := _MOVE1996_OUT; END_IF;
(* RT602_SP Feedback *)
(* RT603_SP Feedback *)
M1_139_003_RT602_SP_FB(bPortKNX := 1, dwIndex_DPT := 139, typDPT := typDPT);
_MOVE2009_OUT := MOVE(EN := M1_139_003_RT602_SP_FB.xUpdate_PLC, IN := M1_139_003_RT602_SP_FB.rValue_OUT, ENO => _MOVE2009_ENO);
IF _MOVE2009_ENO THEN STLV59_563.STLV59_A_563_003.RT602_SP_IN := _MOVE2009_OUT; END_IF;
M1_140_003_RT603_SP_FB(bPortKNX := 1, dwIndex_DPT := 140, typDPT := typDPT);
_MOVE2022_OUT := MOVE(EN := M1_140_003_RT603_SP_FB.xUpdate_PLC, IN := M1_140_003_RT603_SP_FB.rValue_OUT, ENO => _MOVE2022_ENO);
IF _MOVE2022_ENO THEN STLV59_563.STLV59_A_563_003.RT603_SP_IN := _MOVE2022_OUT; END_IF;
(* RT604_SP Feedback *)
(* RT605_SP Feedback *)
M1_141_003_RT604_SP_FB(bPortKNX := 1, dwIndex_DPT := 141, typDPT := typDPT);
_MOVE2035_OUT := MOVE(EN := M1_141_003_RT604_SP_FB.xUpdate_PLC, IN := M1_141_003_RT604_SP_FB.rValue_OUT, ENO => _MOVE2035_ENO);
IF _MOVE2035_ENO THEN STLV59_563.STLV59_A_563_003.RT604_SP_IN := _MOVE2035_OUT; END_IF;
M1_142_003_RT605_SP_FB(bPortKNX := 1, dwIndex_DPT := 142, typDPT := typDPT);
_MOVE2048_OUT := MOVE(EN := M1_142_003_RT605_SP_FB.xUpdate_PLC, IN := M1_142_003_RT605_SP_FB.rValue_OUT, ENO => _MOVE2048_ENO);
IF _MOVE2048_ENO THEN STLV59_563.STLV59_A_563_003.RT605_SP_IN := _MOVE2048_OUT; END_IF;
(* RT606_SP Feedback *)
(* RT607_SP Feedback *)
M1_143_003_RT606_SP_FB(bPortKNX := 1, dwIndex_DPT := 143, typDPT := typDPT);
_MOVE2061_OUT := MOVE(EN := M1_143_003_RT606_SP_FB.xUpdate_PLC, IN := M1_143_003_RT606_SP_FB.rValue_OUT, ENO => _MOVE2061_ENO);
IF _MOVE2061_ENO THEN STLV59_563.STLV59_A_563_003.RT606_SP_IN := _MOVE2061_OUT; END_IF;
M1_144_003_RT607_SP_FB(bPortKNX := 1, dwIndex_DPT := 144, typDPT := typDPT);
_MOVE2074_OUT := MOVE(EN := M1_144_003_RT607_SP_FB.xUpdate_PLC, IN := M1_144_003_RT607_SP_FB.rValue_OUT, ENO => _MOVE2074_ENO);
IF _MOVE2074_ENO THEN STLV59_563.STLV59_A_563_003.RT607_SP_IN := _MOVE2074_OUT; END_IF;
(* RT608_SP Feedback *)
(* RT609_SP Feedback *)
M1_145_003_RT608_SP_FB(bPortKNX := 1, dwIndex_DPT := 145, typDPT := typDPT);
_MOVE2087_OUT := MOVE(EN := M1_145_003_RT608_SP_FB.xUpdate_PLC, IN := M1_145_003_RT608_SP_FB.rValue_OUT, ENO => _MOVE2087_ENO);
IF _MOVE2087_ENO THEN STLV59_563.STLV59_A_563_003.RT608_SP_IN := _MOVE2087_OUT; END_IF;
M1_146_003_RT609_SP_FB(bPortKNX := 1, dwIndex_DPT := 146, typDPT := typDPT);
_MOVE2100_OUT := MOVE(EN := M1_146_003_RT609_SP_FB.xUpdate_PLC, IN := M1_146_003_RT609_SP_FB.rValue_OUT, ENO => _MOVE2100_ENO);
IF _MOVE2100_ENO THEN STLV59_563.STLV59_A_563_003.RT609_SP_IN := _MOVE2100_OUT; END_IF;
(* LU601_V *)
(* LU602_V *)
M1_147_003_LU601_V(bPortKNX := 1, dwIndex_DPT := 147, typDPT := typDPT);
_MOVE2113_OUT := MOVE(EN := M1_147_003_LU601_V.xUpdate_PLC, IN := M1_147_003_LU601_V.xSwitch_OUT, ENO => _MOVE2113_ENO);
IF _MOVE2113_ENO THEN STLV59_563.STLV59_A_563_003.LU601_V := _MOVE2113_OUT; END_IF;
M1_148_003_LU602_V(bPortKNX := 1, dwIndex_DPT := 148, typDPT := typDPT);
_MOVE2126_OUT := MOVE(EN := M1_148_003_LU602_V.xUpdate_PLC, IN := M1_148_003_LU602_V.xSwitch_OUT, ENO => _MOVE2126_ENO);
IF _MOVE2126_ENO THEN STLV59_563.STLV59_A_563_003.LU602_V := _MOVE2126_OUT; END_IF;
(* LU603_V *)
(* LU604_V *)
M1_149_003_LU603_V(bPortKNX := 1, dwIndex_DPT := 149, typDPT := typDPT);
_MOVE2139_OUT := MOVE(EN := M1_149_003_LU603_V.xUpdate_PLC, IN := M1_149_003_LU603_V.xSwitch_OUT, ENO => _MOVE2139_ENO);
IF _MOVE2139_ENO THEN STLV59_563.STLV59_A_563_003.LU603_V := _MOVE2139_OUT; END_IF;
M1_150_003_LU604_V(bPortKNX := 1, dwIndex_DPT := 150, typDPT := typDPT);
_MOVE2152_OUT := MOVE(EN := M1_150_003_LU604_V.xUpdate_PLC, IN := M1_150_003_LU604_V.xSwitch_OUT, ENO => _MOVE2152_ENO);
IF _MOVE2152_ENO THEN STLV59_563.STLV59_A_563_003.LU604_V := _MOVE2152_OUT; END_IF;
(* LU605_V *)
(* LU606_V *)
M1_151_003_LU605_V(bPortKNX := 1, dwIndex_DPT := 151, typDPT := typDPT);
_MOVE2165_OUT := MOVE(EN := M1_151_003_LU605_V.xUpdate_PLC, IN := M1_151_003_LU605_V.xSwitch_OUT, ENO => _MOVE2165_ENO);
IF _MOVE2165_ENO THEN STLV59_563.STLV59_A_563_003.LU605_V := _MOVE2165_OUT; END_IF;
M1_152_003_LU606_V(bPortKNX := 1, dwIndex_DPT := 152, typDPT := typDPT);
_MOVE2178_OUT := MOVE(EN := M1_152_003_LU606_V.xUpdate_PLC, IN := M1_152_003_LU606_V.xSwitch_OUT, ENO => _MOVE2178_ENO);
IF _MOVE2178_ENO THEN STLV59_563.STLV59_A_563_003.LU606_V := _MOVE2178_OUT; END_IF;
(* LU607_V *)
(* LU608_V *)
M1_153_003_LU607_V(bPortKNX := 1, dwIndex_DPT := 153, typDPT := typDPT);
_MOVE2191_OUT := MOVE(EN := M1_153_003_LU607_V.xUpdate_PLC, IN := M1_153_003_LU607_V.xSwitch_OUT, ENO => _MOVE2191_ENO);
IF _MOVE2191_ENO THEN STLV59_563.STLV59_A_563_003.LU607_V := _MOVE2191_OUT; END_IF;
M1_154_003_LU608_V(bPortKNX := 1, dwIndex_DPT := 154, typDPT := typDPT);
_MOVE2204_OUT := MOVE(EN := M1_154_003_LU608_V.xUpdate_PLC, IN := M1_154_003_LU608_V.xSwitch_OUT, ENO => _MOVE2204_ENO);
IF _MOVE2204_ENO THEN STLV59_563.STLV59_A_563_003.LU608_V := _MOVE2204_OUT; END_IF;
(* LU609_V *)
(* LU601_AL *)
M1_155_003_LU609_V(bPortKNX := 1, dwIndex_DPT := 155, typDPT := typDPT);
_MOVE2217_OUT := MOVE(EN := M1_155_003_LU609_V.xUpdate_PLC, IN := M1_155_003_LU609_V.xSwitch_OUT, ENO => _MOVE2217_ENO);
IF _MOVE2217_ENO THEN STLV59_563.STLV59_A_563_003.LU609_V := _MOVE2217_OUT; END_IF;
M1_156_003_LU601_AL(bPortKNX := 1, dwIndex_DPT := 156, typDPT := typDPT);
_MOVE2230_OUT := MOVE(EN := M1_156_003_LU601_AL.xUpdate_PLC, IN := M1_156_003_LU601_AL.xSwitch_OUT, ENO => _MOVE2230_ENO);
IF _MOVE2230_ENO THEN STLV59_563.STLV59_A_563_003.LU601_AL := _MOVE2230_OUT; END_IF;
(* LU602_AL *)
(* LU603_AL *)
M1_157_003_LU602_AL(bPortKNX := 1, dwIndex_DPT := 157, typDPT := typDPT);
_MOVE2243_OUT := MOVE(EN := M1_157_003_LU602_AL.xUpdate_PLC, IN := M1_157_003_LU602_AL.xSwitch_OUT, ENO => _MOVE2243_ENO);
IF _MOVE2243_ENO THEN STLV59_563.STLV59_A_563_003.LU602_AL := _MOVE2243_OUT; END_IF;
M1_158_003_LU603_AL(bPortKNX := 1, dwIndex_DPT := 158, typDPT := typDPT);
_MOVE2256_OUT := MOVE(EN := M1_158_003_LU603_AL.xUpdate_PLC, IN := M1_158_003_LU603_AL.xSwitch_OUT, ENO => _MOVE2256_ENO);
IF _MOVE2256_ENO THEN STLV59_563.STLV59_A_563_003.LU603_AL := _MOVE2256_OUT; END_IF;
(* LU604_AL *)
(* LU605_AL *)
M1_159_003_LU604_AL(bPortKNX := 1, dwIndex_DPT := 159, typDPT := typDPT);
_MOVE2269_OUT := MOVE(EN := M1_159_003_LU604_AL.xUpdate_PLC, IN := M1_159_003_LU604_AL.xSwitch_OUT, ENO => _MOVE2269_ENO);
IF _MOVE2269_ENO THEN STLV59_563.STLV59_A_563_003.LU604_AL := _MOVE2269_OUT; END_IF;
M1_160_003_LU605_AL(bPortKNX := 1, dwIndex_DPT := 160, typDPT := typDPT);
_MOVE2282_OUT := MOVE(EN := M1_160_003_LU605_AL.xUpdate_PLC, IN := M1_160_003_LU605_AL.xSwitch_OUT, ENO => _MOVE2282_ENO);
IF _MOVE2282_ENO THEN STLV59_563.STLV59_A_563_003.LU605_AL := _MOVE2282_OUT; END_IF;
(* LU606_AL *)
(* LU607_AL *)
M1_161_003_LU606_AL(bPortKNX := 1, dwIndex_DPT := 161, typDPT := typDPT);
_MOVE2295_OUT := MOVE(EN := M1_161_003_LU606_AL.xUpdate_PLC, IN := M1_161_003_LU606_AL.xSwitch_OUT, ENO => _MOVE2295_ENO);
IF _MOVE2295_ENO THEN STLV59_563.STLV59_A_563_003.LU606_AL := _MOVE2295_OUT; END_IF;
M1_162_003_LU607_AL(bPortKNX := 1, dwIndex_DPT := 162, typDPT := typDPT);
_MOVE2308_OUT := MOVE(EN := M1_162_003_LU607_AL.xUpdate_PLC, IN := M1_162_003_LU607_AL.xSwitch_OUT, ENO => _MOVE2308_ENO);
IF _MOVE2308_ENO THEN STLV59_563.STLV59_A_563_003.LU607_AL := _MOVE2308_OUT; END_IF;
(* LU608_AL *)
(* LU609_AL *)
M1_163_003_LU608_AL(bPortKNX := 1, dwIndex_DPT := 163, typDPT := typDPT);
_MOVE2321_OUT := MOVE(EN := M1_163_003_LU608_AL.xUpdate_PLC, IN := M1_163_003_LU608_AL.xSwitch_OUT, ENO => _MOVE2321_ENO);
IF _MOVE2321_ENO THEN STLV59_563.STLV59_A_563_003.LU608_AL := _MOVE2321_OUT; END_IF;
M1_164_003_LU609_AL(bPortKNX := 1, dwIndex_DPT := 164, typDPT := typDPT);
_MOVE2334_OUT := MOVE(EN := M1_164_003_LU609_AL.xUpdate_PLC, IN := M1_164_003_LU609_AL.xSwitch_OUT, ENO => _MOVE2334_ENO);
IF _MOVE2334_ENO THEN STLV59_563.STLV59_A_563_003.LU609_AL := _MOVE2334_OUT; END_IF;
(* LU601_CMD *)
(* LU602_CMD *)
M1_165_003_LU601_CMD(bPortKNX := 1, dwIndex_DPT := 165, xSwitch_IN := STLV59_563.STLV59_A_563_003.LU601_CMD, xUpdate_KNX := i = 60, typDPT := typDPT);
M1_166_003_LU602_CMD(bPortKNX := 1, dwIndex_DPT := 166, xSwitch_IN := STLV59_563.STLV59_A_563_003.LU602_CMD, xUpdate_KNX := i = 61, typDPT := typDPT);
(* LU603_CMD *)
(* LU604_CMD *)
M1_167_003_LU603_CMD(bPortKNX := 1, dwIndex_DPT := 167, xSwitch_IN := STLV59_563.STLV59_A_563_003.LU603_CMD, xUpdate_KNX := i = 62, typDPT := typDPT);
M1_168_003_LU604_CMD(bPortKNX := 1, dwIndex_DPT := 168, xSwitch_IN := STLV59_563.STLV59_A_563_003.LU604_CMD, xUpdate_KNX := i = 63, typDPT := typDPT);
(* LU605_CMD *)
(* LU606_CMD *)
M1_169_003_LU605_CMD(bPortKNX := 1, dwIndex_DPT := 169, xSwitch_IN := STLV59_563.STLV59_A_563_003.LU605_CMD, xUpdate_KNX := i = 64, typDPT := typDPT);
M1_170_003_LU606_CMD(bPortKNX := 1, dwIndex_DPT := 170, xSwitch_IN := STLV59_563.STLV59_A_563_003.LU606_CMD, xUpdate_KNX := i = 65, typDPT := typDPT);
(* LU607_CMD *)
(* LU608_CMD *)
M1_171_003_LU607_CMD(bPortKNX := 1, dwIndex_DPT := 171, xSwitch_IN := STLV59_563.STLV59_A_563_003.LU607_CMD, xUpdate_KNX := i = 66, typDPT := typDPT);
M1_172_003_LU608_CMD(bPortKNX := 1, dwIndex_DPT := 172, xSwitch_IN := STLV59_563.STLV59_A_563_003.LU608_CMD, xUpdate_KNX := i = 67, typDPT := typDPT);
(* LU609_CMD *)
(* OPM_001 *)
M1_173_003_LU609_CMD(bPortKNX := 1, dwIndex_DPT := 173, xSwitch_IN := STLV59_563.STLV59_A_563_003.LU609_CMD, xUpdate_KNX := i = 68, typDPT := typDPT);
M1_174_003_OPM_001(bPortKNX := 1, dwIndex_DPT := 174, bIN := STLV59_563.STLV59_A_563_003.OPM_001, xUpdate_KNX := i = 69, typDPT := typDPT);
(* OPM_002 *)
(* OPM_003 *)
M1_175_003_OPM_002(bPortKNX := 1, dwIndex_DPT := 175, bIN := STLV59_563.STLV59_A_563_003.OPM_002, xUpdate_KNX := i = 70, typDPT := typDPT);
M1_176_003_OPM_003(bPortKNX := 1, dwIndex_DPT := 176, bIN := STLV59_563.STLV59_A_563_003.OPM_003, xUpdate_KNX := i = 71, typDPT := typDPT);
(* OPM_004 *)
(* OPM_005 *)
M1_177_003_OPM_004(bPortKNX := 1, dwIndex_DPT := 177, bIN := STLV59_563.STLV59_A_563_003.OPM_004, xUpdate_KNX := i = 72, typDPT := typDPT);
M1_178_003_OPM_005(bPortKNX := 1, dwIndex_DPT := 178, bIN := STLV59_563.STLV59_A_563_003.OPM_005, xUpdate_KNX := i = 73, typDPT := typDPT);
(* OPM_006 *)
(* OPM_007 *)
M1_179_003_OPM_006(bPortKNX := 1, dwIndex_DPT := 179, bIN := STLV59_563.STLV59_A_563_003.OPM_006, xUpdate_KNX := i = 74, typDPT := typDPT);
M1_180_003_OPM_007(bPortKNX := 1, dwIndex_DPT := 180, bIN := STLV59_563.STLV59_A_563_003.OPM_007, xUpdate_KNX := i = 75, typDPT := typDPT);
(* OPM_008 *)
(* OPM_009 *)
M1_181_003_OPM_008(bPortKNX := 1, dwIndex_DPT := 181, bIN := STLV59_563.STLV59_A_563_003.OPM_008, xUpdate_KNX := i = 76, typDPT := typDPT);
M1_182_003_OPM_009(bPortKNX := 1, dwIndex_DPT := 182, bIN := STLV59_563.STLV59_A_563_003.OPM_009, xUpdate_KNX := i = 77, typDPT := typDPT);
END_PROGRAM

PROGRAM PRG_563_Romstyring
  VAR
    Rom_001 : fbRomtype_11111111111111;  (* 001 *)
    Rom_002 : fbRomtype_33333333333333;  (* 002 *)
    Rom_003 : fbRomtype_99999999999999;  (* 003 *)
  END_VAR

(* CFC diagram, written out as Structured Text *)
(* Rom 001 *)
Rom_001(RB601_HVAC := STLV59_563.STLV59_A_563_001.RB601_HVAC, RT601_CT := STLV59_563.STLV59_A_563_001.RT601_CT, RT601_SP_D := STLV59_563.STLV59_A_563_001.RT601_SP_D, RT601_SP_S := STLV59_563.STLV59_A_563_001.RT601_SP_S, RT601_SP_N := STLV59_563.STLV59_A_563_001.RT601_SP_N, RT601_SP_F := STLV59_563.STLV59_A_563_001.RT601_SP_F, OPM := STLV59_563.STLV59_A_563_001.OPM, RY601_CV := STLV59_563.STLV59_A_563_001.RY601_CV, RY601_SP := STLV59_563.STLV59_A_563_001.RY601_SP, LH601_MAN := STLV59_563.STLV59_A_563_001.LH601_MAN, LC601_SP := STLV59_563.STLV59_A_563_001.LC601_SP, LC601_MAN := STLV59_563.STLV59_A_563_001.LC601_MAN, RT601_SP_IN := STLV59_563.STLV59_A_563_001.RT601_SP_IN, LU601_V := STLV59_563.STLV59_A_563_001.LU601_V);
STLV59_563.STLV59_A_563_001.OPM_CV := Rom_001.OPM_CV;
STLV59_563.STLV59_A_563_001.RT601_CS := Rom_001.RT601_CS;
STLV59_563.STLV59_A_563_001.RY601_OP := Rom_001.RY601_OP;
STLV59_563.STLV59_A_563_001.LH601_OP := Rom_001.LH601_OP;
STLV59_563.STLV59_A_563_001.LH601_CMD := Rom_001.LH601_CMD;
STLV59_563.STLV59_A_563_001.LC601_OP := Rom_001.LC601_OP;
STLV59_563.STLV59_A_563_001.LC601_CMD := Rom_001.LC601_CMD;
STLV59_563.STLV59_A_563_001.LU601_CMD := Rom_001.LU601_CMD;
STLV59_563.STLV59_A_563_001.OPM_001 := Rom_001.OPM_001;
(* Rom 002 *)
Rom_002(RB601_HVAC := STLV59_563.STLV59_A_563_002.RB601_HVAC, RB602_HVAC := STLV59_563.STLV59_A_563_002.RB602_HVAC, RB603_HVAC := STLV59_563.STLV59_A_563_002.RB603_HVAC, RT601_CT := STLV59_563.STLV59_A_563_002.RT601_CT, RT602_CT := STLV59_563.STLV59_A_563_002.RT602_CT, RT602_SP := STLV59_563.STLV59_A_563_002.RT602_SP, RT603_CT := STLV59_563.STLV59_A_563_002.RT603_CT, RT603_SP := STLV59_563.STLV59_A_563_002.RT603_SP, RT601_SP_D := STLV59_563.STLV59_A_563_002.RT601_SP_D, RT601_SP_S := STLV59_563.STLV59_A_563_002.RT601_SP_S, RT601_SP_N := STLV59_563.STLV59_A_563_002.RT601_SP_N, RT601_SP_F := STLV59_563.STLV59_A_563_002.RT601_SP_F, OPM := STLV59_563.STLV59_A_563_002.OPM, RY601_CV := STLV59_563.STLV59_A_563_002.RY601_CV, RY602_CV := STLV59_563.STLV59_A_563_002.RY602_CV, RY603_CV := STLV59_563.STLV59_A_563_002.RY603_CV, RY601_SP := STLV59_563.STLV59_A_563_002.RY601_SP, LH601_MAN := STLV59_563.STLV59_A_563_002.LH601_MAN, LC601_SP := STLV59_563.STLV59_A_563_002.LC601_SP, LC601_MAN := STLV59_563.STLV59_A_563_002.LC601_MAN, RT601_SP_IN := STLV59_563.STLV59_A_563_002.RT601_SP_IN, RT602_SP_IN := STLV59_563.STLV59_A_563_002.RT602_SP_IN, RT603_SP_IN := STLV59_563.STLV59_A_563_002.RT603_SP_IN, LU601_V := STLV59_563.STLV59_A_563_002.LU601_V, LU602_V := STLV59_563.STLV59_A_563_002.LU602_V, LU603_V := STLV59_563.STLV59_A_563_002.LU603_V);
STLV59_563.STLV59_A_563_002.OPM_CV := Rom_002.OPM_CV;
STLV59_563.STLV59_A_563_002.RT601_CS := Rom_002.RT601_CS;
STLV59_563.STLV59_A_563_002.RY601_OP := Rom_002.RY601_OP;
STLV59_563.STLV59_A_563_002.LH601_OP := Rom_002.LH601_OP;
STLV59_563.STLV59_A_563_002.LH602_OP := Rom_002.LH602_OP;
STLV59_563.STLV59_A_563_002.LH603_OP := Rom_002.LH603_OP;
STLV59_563.STLV59_A_563_002.LH601_CMD := Rom_002.LH601_CMD;
STLV59_563.STLV59_A_563_002.LH602_CMD := Rom_002.LH602_CMD;
STLV59_563.STLV59_A_563_002.LH603_CMD := Rom_002.LH603_CMD;
STLV59_563.STLV59_A_563_002.LC601_OP := Rom_002.LC601_OP;
STLV59_563.STLV59_A_563_002.LC602_OP := Rom_002.LC602_OP;
STLV59_563.STLV59_A_563_002.LC603_OP := Rom_002.LC603_OP;
STLV59_563.STLV59_A_563_002.LC601_CMD := Rom_002.LC601_CMD;
STLV59_563.STLV59_A_563_002.LC602_CMD := Rom_002.LC602_CMD;
STLV59_563.STLV59_A_563_002.LC603_CMD := Rom_002.LC603_CMD;
STLV59_563.STLV59_A_563_002.LU601_CMD := Rom_002.LU601_CMD;
STLV59_563.STLV59_A_563_002.LU602_CMD := Rom_002.LU602_CMD;
STLV59_563.STLV59_A_563_002.LU603_CMD := Rom_002.LU603_CMD;
STLV59_563.STLV59_A_563_002.OPM_001 := Rom_002.OPM_001;
STLV59_563.STLV59_A_563_002.OPM_002 := Rom_002.OPM_002;
STLV59_563.STLV59_A_563_002.OPM_003 := Rom_002.OPM_003;
(* Rom 003 *)
Rom_003(RB601_HVAC := STLV59_563.STLV59_A_563_003.RB601_HVAC, RB602_HVAC := STLV59_563.STLV59_A_563_003.RB602_HVAC, RB603_HVAC := STLV59_563.STLV59_A_563_003.RB603_HVAC, RB604_HVAC := STLV59_563.STLV59_A_563_003.RB604_HVAC, RB605_HVAC := STLV59_563.STLV59_A_563_003.RB605_HVAC, RB606_HVAC := STLV59_563.STLV59_A_563_003.RB606_HVAC, RB607_HVAC := STLV59_563.STLV59_A_563_003.RB607_HVAC, RB608_HVAC := STLV59_563.STLV59_A_563_003.RB608_HVAC, RB609_HVAC := STLV59_563.STLV59_A_563_003.RB609_HVAC, RT601_CT := STLV59_563.STLV59_A_563_003.RT601_CT, RT602_CT := STLV59_563.STLV59_A_563_003.RT602_CT, RT602_SP := STLV59_563.STLV59_A_563_003.RT602_SP, RT603_CT := STLV59_563.STLV59_A_563_003.RT603_CT, RT603_SP := STLV59_563.STLV59_A_563_003.RT603_SP, RT604_CT := STLV59_563.STLV59_A_563_003.RT604_CT, RT604_SP := STLV59_563.STLV59_A_563_003.RT604_SP, RT605_CT := STLV59_563.STLV59_A_563_003.RT605_CT, RT605_SP := STLV59_563.STLV59_A_563_003.RT605_SP, RT606_CT := STLV59_563.STLV59_A_563_003.RT606_CT, RT606_SP := STLV59_563.STLV59_A_563_003.RT606_SP, RT607_CT := STLV59_563.STLV59_A_563_003.RT607_CT, RT607_SP := STLV59_563.STLV59_A_563_003.RT607_SP, RT608_CT := STLV59_563.STLV59_A_563_003.RT608_CT, RT608_SP := STLV59_563.STLV59_A_563_003.RT608_SP, RT609_CT := STLV59_563.STLV59_A_563_003.RT609_CT, RT609_SP := STLV59_563.STLV59_A_563_003.RT609_SP, RT601_SP_D := STLV59_563.STLV59_A_563_003.RT601_SP_D, RT601_SP_S := STLV59_563.STLV59_A_563_003.RT601_SP_S, RT601_SP_N := STLV59_563.STLV59_A_563_003.RT601_SP_N, RT601_SP_F := STLV59_563.STLV59_A_563_003.RT601_SP_F, OPM := STLV59_563.STLV59_A_563_003.OPM, RY601_CV := STLV59_563.STLV59_A_563_003.RY601_CV, RY602_CV := STLV59_563.STLV59_A_563_003.RY602_CV, RY603_CV := STLV59_563.STLV59_A_563_003.RY603_CV, RY604_CV := STLV59_563.STLV59_A_563_003.RY604_CV, RY605_CV := STLV59_563.STLV59_A_563_003.RY605_CV, RY606_CV := STLV59_563.STLV59_A_563_003.RY606_CV, RY607_CV := STLV59_563.STLV59_A_563_003.RY607_CV, RY608_CV := STLV59_563.STLV59_A_563_003.RY608_CV, RY609_CV := STLV59_563.STLV59_A_563_003.RY609_CV, RY601_SP := STLV59_563.STLV59_A_563_003.RY601_SP, LH601_MAN := STLV59_563.STLV59_A_563_003.LH601_MAN, LC601_SP := STLV59_563.STLV59_A_563_003.LC601_SP, LC601_MAN := STLV59_563.STLV59_A_563_003.LC601_MAN, RT601_SP_IN := STLV59_563.STLV59_A_563_003.RT601_SP_IN, RT602_SP_IN := STLV59_563.STLV59_A_563_003.RT602_SP_IN, RT603_SP_IN := STLV59_563.STLV59_A_563_003.RT603_SP_IN, RT604_SP_IN := STLV59_563.STLV59_A_563_003.RT604_SP_IN, RT605_SP_IN := STLV59_563.STLV59_A_563_003.RT605_SP_IN, RT606_SP_IN := STLV59_563.STLV59_A_563_003.RT606_SP_IN, RT607_SP_IN := STLV59_563.STLV59_A_563_003.RT607_SP_IN, RT608_SP_IN := STLV59_563.STLV59_A_563_003.RT608_SP_IN, RT609_SP_IN := STLV59_563.STLV59_A_563_003.RT609_SP_IN, LU601_V := STLV59_563.STLV59_A_563_003.LU601_V, LU602_V := STLV59_563.STLV59_A_563_003.LU602_V, LU603_V := STLV59_563.STLV59_A_563_003.LU603_V, LU604_V := STLV59_563.STLV59_A_563_003.LU604_V, LU605_V := STLV59_563.STLV59_A_563_003.LU605_V, LU606_V := STLV59_563.STLV59_A_563_003.LU606_V, LU607_V := STLV59_563.STLV59_A_563_003.LU607_V, LU608_V := STLV59_563.STLV59_A_563_003.LU608_V, LU609_V := STLV59_563.STLV59_A_563_003.LU609_V);
STLV59_563.STLV59_A_563_003.OPM_CV := Rom_003.OPM_CV;
STLV59_563.STLV59_A_563_003.RT601_CS := Rom_003.RT601_CS;
STLV59_563.STLV59_A_563_003.RY601_OP := Rom_003.RY601_OP;
STLV59_563.STLV59_A_563_003.LH601_OP := Rom_003.LH601_OP;
STLV59_563.STLV59_A_563_003.LH602_OP := Rom_003.LH602_OP;
STLV59_563.STLV59_A_563_003.LH603_OP := Rom_003.LH603_OP;
STLV59_563.STLV59_A_563_003.LH604_OP := Rom_003.LH604_OP;
STLV59_563.STLV59_A_563_003.LH605_OP := Rom_003.LH605_OP;
STLV59_563.STLV59_A_563_003.LH606_OP := Rom_003.LH606_OP;
STLV59_563.STLV59_A_563_003.LH607_OP := Rom_003.LH607_OP;
STLV59_563.STLV59_A_563_003.LH608_OP := Rom_003.LH608_OP;
STLV59_563.STLV59_A_563_003.LH609_OP := Rom_003.LH609_OP;
STLV59_563.STLV59_A_563_003.LH601_CMD := Rom_003.LH601_CMD;
STLV59_563.STLV59_A_563_003.LH602_CMD := Rom_003.LH602_CMD;
STLV59_563.STLV59_A_563_003.LH603_CMD := Rom_003.LH603_CMD;
STLV59_563.STLV59_A_563_003.LH604_CMD := Rom_003.LH604_CMD;
STLV59_563.STLV59_A_563_003.LH605_CMD := Rom_003.LH605_CMD;
STLV59_563.STLV59_A_563_003.LH606_CMD := Rom_003.LH606_CMD;
STLV59_563.STLV59_A_563_003.LH607_CMD := Rom_003.LH607_CMD;
STLV59_563.STLV59_A_563_003.LH608_CMD := Rom_003.LH608_CMD;
STLV59_563.STLV59_A_563_003.LH609_CMD := Rom_003.LH609_CMD;
STLV59_563.STLV59_A_563_003.LC601_OP := Rom_003.LC601_OP;
STLV59_563.STLV59_A_563_003.LC602_OP := Rom_003.LC602_OP;
STLV59_563.STLV59_A_563_003.LC603_OP := Rom_003.LC603_OP;
STLV59_563.STLV59_A_563_003.LC604_OP := Rom_003.LC604_OP;
STLV59_563.STLV59_A_563_003.LC605_OP := Rom_003.LC605_OP;
STLV59_563.STLV59_A_563_003.LC606_OP := Rom_003.LC606_OP;
STLV59_563.STLV59_A_563_003.LC607_OP := Rom_003.LC607_OP;
STLV59_563.STLV59_A_563_003.LC608_OP := Rom_003.LC608_OP;
STLV59_563.STLV59_A_563_003.LC609_OP := Rom_003.LC609_OP;
STLV59_563.STLV59_A_563_003.LC601_CMD := Rom_003.LC601_CMD;
STLV59_563.STLV59_A_563_003.LC602_CMD := Rom_003.LC602_CMD;
STLV59_563.STLV59_A_563_003.LC603_CMD := Rom_003.LC603_CMD;
STLV59_563.STLV59_A_563_003.LC604_CMD := Rom_003.LC604_CMD;
STLV59_563.STLV59_A_563_003.LC605_CMD := Rom_003.LC605_CMD;
STLV59_563.STLV59_A_563_003.LC606_CMD := Rom_003.LC606_CMD;
STLV59_563.STLV59_A_563_003.LC607_CMD := Rom_003.LC607_CMD;
STLV59_563.STLV59_A_563_003.LC608_CMD := Rom_003.LC608_CMD;
STLV59_563.STLV59_A_563_003.LC609_CMD := Rom_003.LC609_CMD;
STLV59_563.STLV59_A_563_003.LU601_CMD := Rom_003.LU601_CMD;
STLV59_563.STLV59_A_563_003.LU602_CMD := Rom_003.LU602_CMD;
STLV59_563.STLV59_A_563_003.LU603_CMD := Rom_003.LU603_CMD;
STLV59_563.STLV59_A_563_003.LU604_CMD := Rom_003.LU604_CMD;
STLV59_563.STLV59_A_563_003.LU605_CMD := Rom_003.LU605_CMD;
STLV59_563.STLV59_A_563_003.LU606_CMD := Rom_003.LU606_CMD;
STLV59_563.STLV59_A_563_003.LU607_CMD := Rom_003.LU607_CMD;
STLV59_563.STLV59_A_563_003.LU608_CMD := Rom_003.LU608_CMD;
STLV59_563.STLV59_A_563_003.LU609_CMD := Rom_003.LU609_CMD;
STLV59_563.STLV59_A_563_003.OPM_001 := Rom_003.OPM_001;
STLV59_563.STLV59_A_563_003.OPM_002 := Rom_003.OPM_002;
STLV59_563.STLV59_A_563_003.OPM_003 := Rom_003.OPM_003;
STLV59_563.STLV59_A_563_003.OPM_004 := Rom_003.OPM_004;
STLV59_563.STLV59_A_563_003.OPM_005 := Rom_003.OPM_005;
STLV59_563.STLV59_A_563_003.OPM_006 := Rom_003.OPM_006;
STLV59_563.STLV59_A_563_003.OPM_007 := Rom_003.OPM_007;
STLV59_563.STLV59_A_563_003.OPM_008 := Rom_003.OPM_008;
STLV59_563.STLV59_A_563_003.OPM_009 := Rom_003.OPM_009;
END_PROGRAM

PROGRAM PRG_360_HVAC

	STLV59_563.STLV59_A_563_RB001_HVAC:=
(
	STLV59_563.STLV59_A_563_001.RB601_HVAC OR
	STLV59_563.STLV59_A_563_002.RB601_HVAC OR
	STLV59_563.STLV59_A_563_002.RB602_HVAC OR
	STLV59_563.STLV59_A_563_002.RB603_HVAC OR
	STLV59_563.STLV59_A_563_003.RB601_HVAC OR
	STLV59_563.STLV59_A_563_003.RB602_HVAC OR
	STLV59_563.STLV59_A_563_003.RB603_HVAC OR
	STLV59_563.STLV59_A_563_003.RB604_HVAC OR
	STLV59_563.STLV59_A_563_003.RB605_HVAC OR
	STLV59_563.STLV59_A_563_003.RB606_HVAC OR
	STLV59_563.STLV59_A_563_003.RB607_HVAC OR
	STLV59_563.STLV59_A_563_003.RB608_HVAC OR
	STLV59_563.STLV59_A_563_003.RB609_HVAC
);
END_PROGRAM
